(* CoDeSys 2.3 library: GermesLib_1_2.lib *)
(* Libraries: PID_Regulators.lib 6.11.19 15:29:27, Util.lib 18.5.10 15:14:28, STANDARD.LIB 4.10.05 11:14:46, IECSFC.LIB 13.4.06 15:51:28, ANALYZATION.LIB 5.10.99 09:05:06 *)

(* POU ChoosePumpRegime, CFC *)
FUNCTION_BLOCK ChoosePumpRegime
VAR
	pump1RStrig: RS;		(*Триггер-защелка выбора режима с главным первым насосом.*)
	pump2RStrig: RS;		(*Триггер-защелка выбора режима с главным вторым насосом.*)
	byCounterRStrig: RS;		(*Триггер-защелка выбора режима с запуском по количеству включений.*)
	byWorkTimeRStrig: RS;		(*Триггер-защелка выбора режима с запуском по наработке.*)
	Pump1MainDetector: R_TRIG;		(*Детектор переднего фронта включения режима, когда главный насос - первый.
Для сброса остальных значений.*)
	Pump2MainDetector: R_TRIG;		(*Детектор переднего фронта включения режима, когда главный насос - второй.
Для сброса остальных значений.*)
	ByCounterDetector: R_TRIG;		(*Детектор переднего фронта включения режима по количеству включений.
Для сброса остальных значений.*)
	ByWorkTimeDetector: R_TRIG;		(*Детектор переднего фронта включения режима по наработке.
Для сброса остальных значений.*)
END_VAR
VAR_INPUT
	start: BOOL;		(*Сигнал на включение насоса.
Активируется выход согласно выбранного режима.*)
	pump1Main: BOOL;		(*Режим: первый насос главный, второй - резервный.
Включать импульсом. Включать импульсом.*)
	pump2Main: BOOL;		(*Режим: второй насос главный, первый - резервный.
Включать импульсом. Включать импульсом.*)
	byCounter: BOOL;		(*Режим: запуск по количеству включений.
Включится с меньшим количеством стартов. Включать импульсом.*)
	byWorkTime: BOOL;		(*Режим: запуск по наработке.
Включится насос с меньшей наработкой. Включать импульсом.*)
END_VAR
VAR_OUTPUT
	pump1MainActive: BOOL;		(*Активный режим: первый насос главный.*)
	pump2MainActive: BOOL;		(*Активный режим: второй насос главный.*)
	byCounterActive: BOOL;		(*Активный режим: включение по количеству запусков.*)
	byWorkTimeActive: BOOL;		(*Активный режим: по наработке.*)
	startPump1: BOOL;		(*Запуск первого насоса как главного (основного).*)
	startPump2: BOOL;		(*Запуск второго насоса как главного (основного).*)
	startByCounter: BOOL;		(*Запуск насоса по количеству стартов.
			Запустится с меньшим. Если одинаково, то - первый.*)
	startByWorkTime: BOOL;		(*Запуск по наработке.
			Включится с меньшей. Если одинаково, то - первый.*)
END_VAR
VAR (* helpers for the ST form of the networks *)
	_en62 : BOOL;
	_t62 : BOOL;
	_en72 : BOOL;
	_t72 : BOOL;
	_en78 : BOOL;
	_t78 : BOOL;
	_en84 : BOOL;
	_t84 : BOOL;
END_VAR
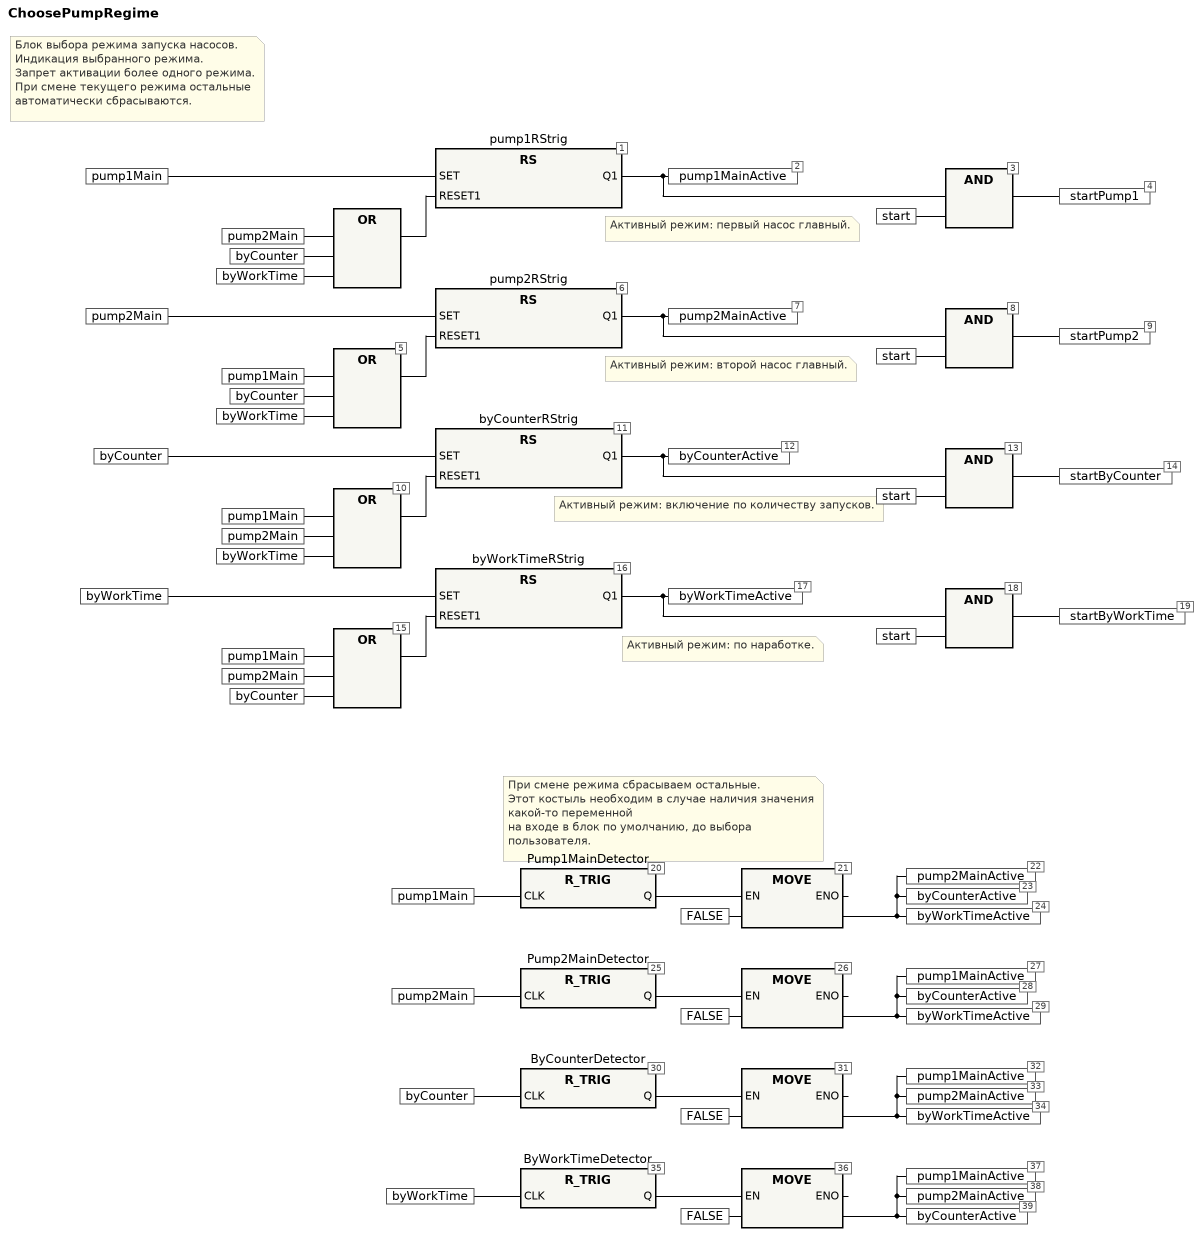
_CFC_ (* Continuous Function Chart, elements in execution order *)
(* При смене режима сбрасываем остальные. / Этот костыль необходим в случае наличия значения какой-то переменной / на входе в блок по умолчанию, до выбора пользователя. *)
(* Активный режим: второй насос главный. *)
(* Активный режим: по наработке. *)
(* Активный режим: включение по количеству запусков. *)
(* Активный режим: первый насос главный. *)
(* Блок выбора режима запуска насосов. / Индикация выбранного режима. / Запрет активации более одного режима. / При смене текущего режима остальные автоматически сбрасываются. *)
#0 OR(pump2Main, byCounter, byWorkTime)
#1 pump1RStrig:RS(SET: pump1Main, RESET1: #0)
#2 pump1MainActive <= #1.Q1
#3 AND(#1.Q1, start)
#4 startPump1 <= #3
#5 OR(pump1Main, byCounter, byWorkTime)
#6 pump2RStrig:RS(SET: pump2Main, RESET1: #5)
#7 pump2MainActive <= #6.Q1
#8 AND(#6.Q1, start)
#9 startPump2 <= #8
#10 OR(pump1Main, pump2Main, byWorkTime)
#11 byCounterRStrig:RS(SET: byCounter, RESET1: #10)
#12 byCounterActive <= #11.Q1
#13 AND(#11.Q1, start)
#14 startByCounter <= #13
#15 OR(pump1Main, pump2Main, byCounter)
#16 byWorkTimeRStrig:RS(SET: byWorkTime, RESET1: #15)
#17 byWorkTimeActive <= #16.Q1
#18 AND(#16.Q1, start)
#19 startByWorkTime <= #18
#20 Pump1MainDetector:R_TRIG(CLK: pump1Main)
#21 MOVE(EN: #20.Q, FALSE)
#22 pump2MainActive <= #21
#23 byCounterActive <= #21
#24 byWorkTimeActive <= #21
#25 Pump2MainDetector:R_TRIG(CLK: pump2Main)
#26 MOVE(EN: #25.Q, FALSE)
#27 pump1MainActive <= #26
#28 byCounterActive <= #26
#29 byWorkTimeActive <= #26
#30 ByCounterDetector:R_TRIG(CLK: byCounter)
#31 MOVE(EN: #30.Q, FALSE)
#32 pump1MainActive <= #31
#33 pump2MainActive <= #31
#34 byWorkTimeActive <= #31
#35 ByWorkTimeDetector:R_TRIG(CLK: byWorkTime)
#36 MOVE(EN: #35.Q, FALSE)
#37 pump1MainActive <= #36
#38 pump2MainActive <= #36
#39 byCounterActive <= #36
_END_CFC_
(* the same logic as Structured Text *)
(* При смене режима сбрасываем остальные. / Этот костыль необходим в случае наличия значения какой-то переменной / на входе в блок по умолчанию, до выбора пользователя. *)
(* Активный режим: второй насос главный. *)
(* Активный режим: по наработке. *)
(* Активный режим: включение по количеству запусков. *)
(* Активный режим: первый насос главный. *)
(* Блок выбора режима запуска насосов. / Индикация выбранного режима. / Запрет активации более одного режима. / При смене текущего режима остальные автоматически сбрасываются. *)
pump1RStrig(SET := pump1Main, RESET1 := pump2Main OR byCounter OR byWorkTime);
pump1MainActive := pump1RStrig.Q1;
startPump1 := pump1RStrig.Q1 AND start;
pump2RStrig(SET := pump2Main, RESET1 := pump1Main OR byCounter OR byWorkTime);
pump2MainActive := pump2RStrig.Q1;
startPump2 := pump2RStrig.Q1 AND start;
byCounterRStrig(SET := byCounter, RESET1 := pump1Main OR pump2Main OR byWorkTime);
byCounterActive := byCounterRStrig.Q1;
startByCounter := byCounterRStrig.Q1 AND start;
byWorkTimeRStrig(SET := byWorkTime, RESET1 := pump1Main OR pump2Main OR byCounter);
byWorkTimeActive := byWorkTimeRStrig.Q1;
startByWorkTime := byWorkTimeRStrig.Q1 AND start;
Pump1MainDetector(CLK := pump1Main);
_en62 := Pump1MainDetector.Q;
IF _en62 THEN _t62 := FALSE; END_IF;
IF _en62 THEN pump2MainActive := _t62; END_IF;
IF _en62 THEN byCounterActive := _t62; END_IF;
IF _en62 THEN byWorkTimeActive := _t62; END_IF;
Pump2MainDetector(CLK := pump2Main);
_en72 := Pump2MainDetector.Q;
IF _en72 THEN _t72 := FALSE; END_IF;
IF _en72 THEN pump1MainActive := _t72; END_IF;
IF _en72 THEN byCounterActive := _t72; END_IF;
IF _en72 THEN byWorkTimeActive := _t72; END_IF;
ByCounterDetector(CLK := byCounter);
_en78 := ByCounterDetector.Q;
IF _en78 THEN _t78 := FALSE; END_IF;
IF _en78 THEN pump1MainActive := _t78; END_IF;
IF _en78 THEN pump2MainActive := _t78; END_IF;
IF _en78 THEN byWorkTimeActive := _t78; END_IF;
ByWorkTimeDetector(CLK := byWorkTime);
_en84 := ByWorkTimeDetector.Q;
IF _en84 THEN _t84 := FALSE; END_IF;
IF _en84 THEN pump1MainActive := _t84; END_IF;
IF _en84 THEN pump2MainActive := _t84; END_IF;
IF _en84 THEN byCounterActive := _t84; END_IF;
END_FUNCTION_BLOCK

(* POU ControlAI, CFC *)
FUNCTION_BLOCK ControlAI
VAR_INPUT
	in: REAL;		(*Входное значение.*)
	minValue: REAL := 0;		(*Минимальное значение на выходе при 4мА на входе.
Если ко входу ничего не подключено, то 0.*)
	maxValue: REAL;		(*Максимальное значение на выходе при 20мА на входе.*)
END_VAR
VAR_OUTPUT
	out: REAL;		(*Выходное отфильтрованное значение.*)
	error: BOOL;		(*Ошибка входа.*)
END_VAR
VAR
	LIN_TRAFO: LIN_TRAFO;		(*Блок масштабирования входной величины.*)
	FilterREAL: FilterREAL;		(*Модуль фильтрации сигнала типа REAL.*)
END_VAR
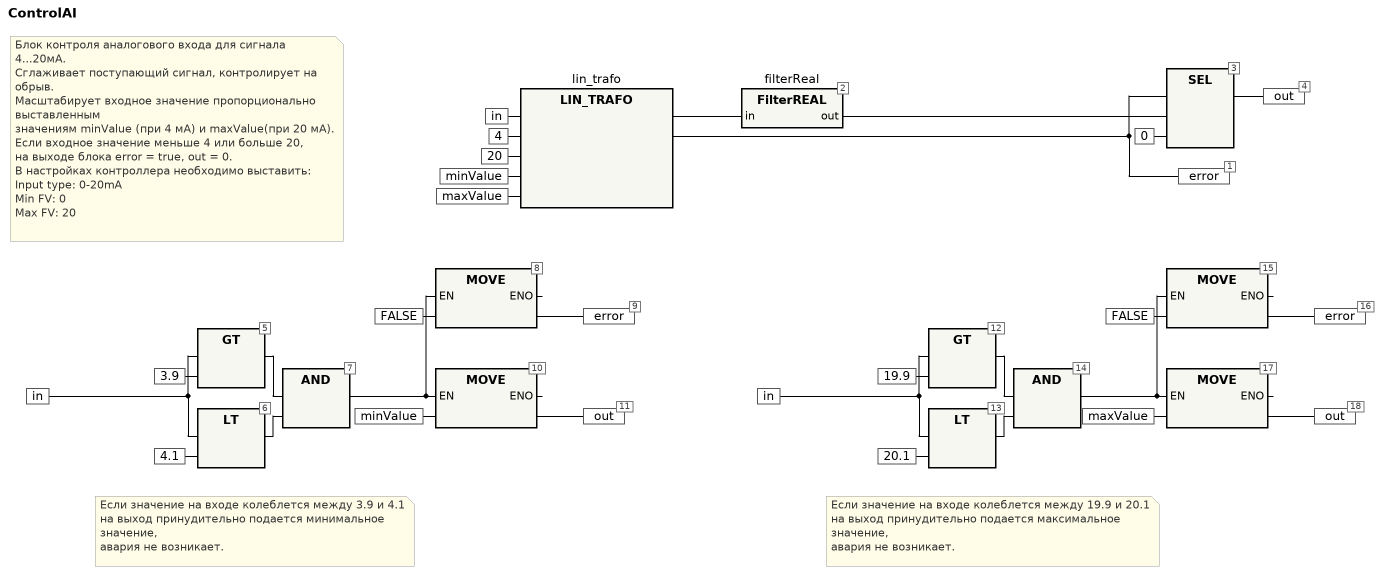
_CFC_ (* Continuous Function Chart, elements in execution order *)
(* Если значение на входе колеблется между 19.9 и 20.1 / на выход принудительно подается максимальное значение, / авария не возникает. *)
(* Если значение на входе колеблется между 3.9 и 4.1 / на выход принудительно подается минимальное значение, / авария не возникает. *)
(* Блок контроля аналогового входа для сигнала 4...20мА. / Сглаживает поступающий сигнал, контролирует на обрыв. / Масштабирует входное значение пропорционально выставленным / значениям minValue (при 4 мА) и maxValue(при 20 мА). / Если входное значение меньше 4 или больше 20, / на выходе блока error = true, out = 0. / В настройках контроллера необходимо выставить: / Input type: 0-20mA / Min FV: 0 / Max FV: 20 *)
#0 lin_trafo:LIN_TRAFO(in, 4, 20, minValue, maxValue)
#1 error <= #0.out 2
#2 filterReal:FilterREAL(in: #0.out 1)
#3 SEL(#0.out 2, #2.out, 0)
#4 out <= #3
#5 GT(in, 3.9)
#6 LT(in, 4.1)
#7 AND(#5, #6)
#8 MOVE(EN: #7, FALSE)
#9 error <= #8
#10 MOVE(EN: #7, minValue)
#11 out <= #10
#12 GT(in, 19.9)
#13 LT(in, 20.1)
#14 AND(#12, #13)
#15 MOVE(EN: #14, FALSE)
#16 error <= #15
#17 MOVE(EN: #14, maxValue)
#18 out <= #17
_END_CFC_
END_FUNCTION_BLOCK

(* POU FilterREAL, ST *)
FUNCTION_BLOCK FilterREAL
VAR_INPUT
	in: REAL; (*Входное значение*)
END_VAR
VAR_OUTPUT
	out: REAL; (*Выходное значение*)
END_VAR
VAR
	k: REAL; (*Коэффициент фильтра.Чем меньше тем плавнее, чем больше, тем быстрее работает фильтр.*)
END_VAR
(*Если разница между входом и выходом больше 0,5, то коэффициент большой, фильтр - быстрый, сглаживание - минимально.*)
IF ABS(in - out) > 0.01 THEN
	k := 0.9;
ELSE
	k:=0.0001;
END_IF
out := (in - out) * k + out;
END_FUNCTION_BLOCK

(* POU CounterManager, CFC *)
FUNCTION_BLOCK CounterManager

VAR
	pump1startsCounter: ImpulsCounter;		(*Счетчик количества включений насоса 1.*)
	pump2startsCounter: ImpulsCounter;		(*Счетчик количества включений насоса 2.*)
	counterRtrig: R_TRIG;		(*Детектор переднего фронта сигнала на запуск.*)
	counterFtrig: F_TRIG;		(*Детектор спада сигнала на запуск.*)
	counterRStrigPump1: RS;		(*RSтриггер сигнала на запуск насоса 1.*)
	counterRStrigPump2: RS;		(*RSтриггер сигнала на запуск насоса 2.*)
END_VAR
VAR_INPUT
	counterStart: BOOL;		(*Сигнал на запуск насоса с наименьшей наработкой.*)
	pump1ON: BOOL;		(*Сигнал подтверждение о запуске насоса 1.*)
	pump2ON: BOOL;		(*Сигнал подтверждение о запуске насоса 2.*)
	Pump1ResetCounter: BOOL;		(*Сброс счетчика включений насоса 1.*)
	Pump2ResetCounter: BOOL;		(*Сброс счетчика включений насоса 2.*)
END_VAR
VAR_OUTPUT
	counterPump1ON: BOOL;		(*Сигнал на запуск насоса 1.*)
	counterPump2ON: BOOL;		(*Сигнал на запуск насоса 2.*)
	counterPump1: DWORD;		(*Количество включений насоса 1.*)
	counterPump2: DWORD;		(*Количество включений насоса 2.*)
END_VAR
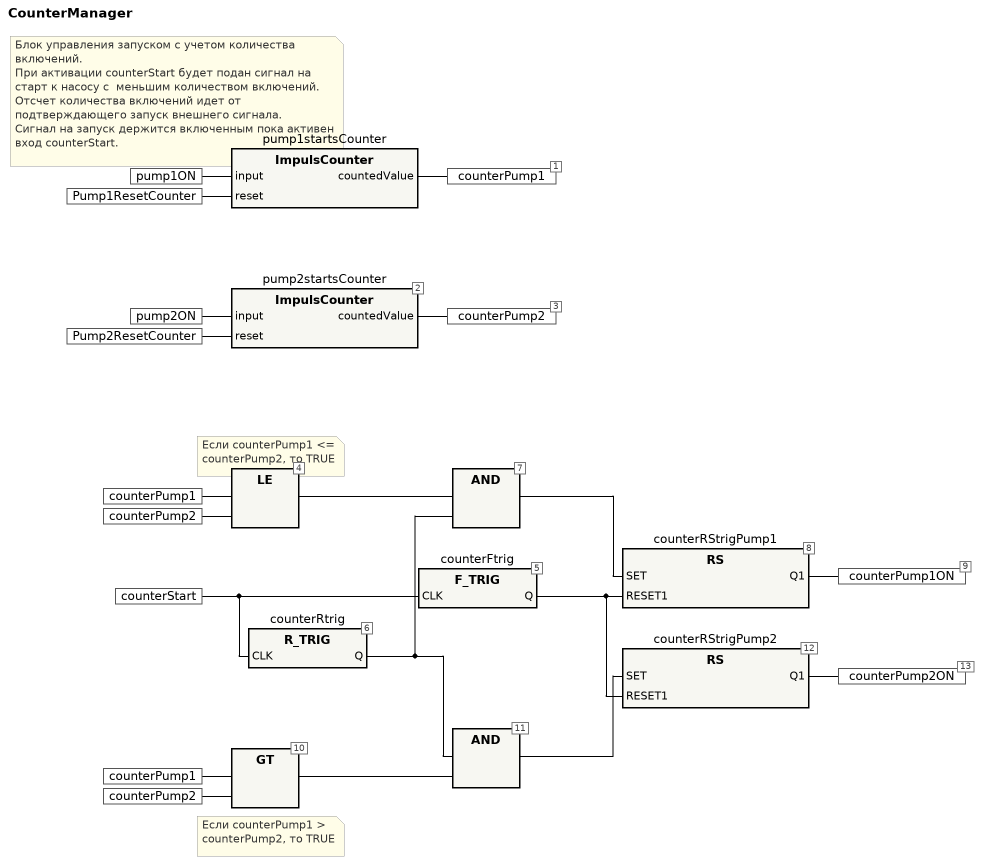
_CFC_ (* Continuous Function Chart, elements in execution order *)
(* Блок управления запуском с учетом количества включений. / При активации counterStart будет подан сигнал на старт к насосу с  меньшим количеством включений. / Отсчет количества включений идет от подтверждающего запуск внешнего сигнала. / Сигнал на запуск держится включенным пока активен вход counterStart. *)
(* Если counterPump1 <= / counterPump2, то TRUE *)
(* Если counterPump1 > / counterPump2, то TRUE *)
#0 pump1startsCounter:ImpulsCounter(input: pump1ON, reset: Pump1ResetCounter)
#1 counterPump1 <= #0.countedValue
#2 pump2startsCounter:ImpulsCounter(input: pump2ON, reset: Pump2ResetCounter)
#3 counterPump2 <= #2.countedValue
#4 LE(counterPump1, counterPump2)
#5 counterFtrig:F_TRIG(CLK: counterStart)
#6 counterRtrig:R_TRIG(CLK: counterStart)
#7 AND(#4, #6.Q)
#8 counterRStrigPump1:RS(SET: #7, RESET1: #5.Q)
#9 counterPump1ON <= #8.Q1
#10 GT(counterPump1, counterPump2)
#11 AND(#6.Q, #10)
#12 counterRStrigPump2:RS(SET: #11, RESET1: #5.Q)
#13 counterPump2ON <= #12.Q1
_END_CFC_
END_FUNCTION_BLOCK

(* POU ImpulsCounter, CFC *)
FUNCTION_BLOCK ImpulsCounter
VAR
	ImpulsDetector: R_TRIG;		(*Триггер переднего фронта входящего импульса.*)
END_VAR
VAR_INPUT
	input: BOOL;		(*Вход для импульсов, которые надо сосчитать.*)
	reset: BOOL;		(*Сброс счетчика.*)
END_VAR
VAR_OUTPUT
	countedValue: DWORD;		(*Суммарное количество импульсов.*)
END_VAR
VAR (* helpers for the ST form of the networks *)
	_t8 : DWORD;
END_VAR
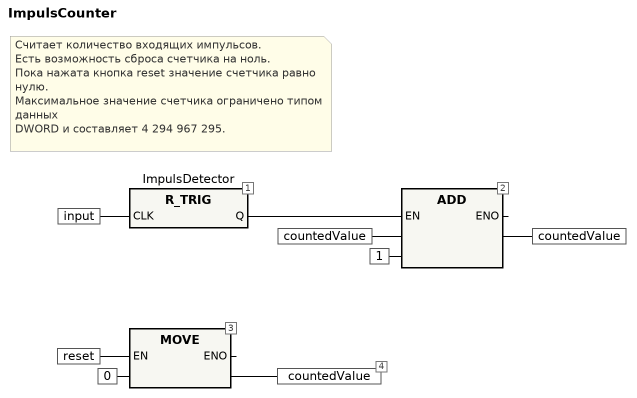
_CFC_ (* Continuous Function Chart, elements in execution order *)
(* Считает количество входящих импульсов. / Есть возможность сброса счетчика на ноль. / Пока нажата кнопка reset значение счетчика равно нулю. / Максимальное значение счетчика ограничено типом данных / DWORD и составляет 4 294 967 295. *)
#0 countedValue <= #2
#1 ImpulsDetector:R_TRIG(CLK: input)
#2 ADD(EN: #1.Q, countedValue, 1)
#3 MOVE(EN: reset, 0)
#4 countedValue <= #3
_END_CFC_
(* the same logic as Structured Text *)
(* Считает количество входящих импульсов. / Есть возможность сброса счетчика на ноль. / Пока нажата кнопка reset значение счетчика равно нулю. / Максимальное значение счетчика ограничено типом данных / DWORD и составляет 4 294 967 295. *)
countedValue := _t8;
ImpulsDetector(CLK := input);
IF ImpulsDetector.Q THEN _t8 := countedValue + 1; END_IF;
IF reset THEN countedValue := 0; END_IF;
END_FUNCTION_BLOCK

(* POU DosingPumpProportional, CFC *)
FUNCTION_BLOCK DosingPumpProportional
VAR_INPUT
	flowValue: REAL;		(*текущее значение мгновенного расхода, кубометров в час.*)
	setMinPumpDosingValue: REAL := 0;		(*задание минимальной производительности доз.насоса.
По умолчанию, если ничего не подключено ко входу, равно нулю.*)
	setMaxPumpDosingValue: REAL;		(*задание максимальной производительности доз.насоса, в мл/мин*)
	minOutputValue: REAL := 4;		(*минимальное значение выходного сигнала.
По умолчанию, если ничего не подключено ко входу, равно 4.*)
	maxOutputValue: REAL := 20;		(*Максимально значение выходного сигнала.
По умолчанию, если ничего не подключено ко входу, равно 20.*)
	setKoeffProportionality: REAL;		(*Задание мл на кубометр (коэф.пропорциональности между расходом и дозированием)*)
	minFlowToStart: REAL := 10;		(*Минимальное значение расхода для подачи сигнала на начало дозирования.
По умолчанию, если ничего не подключено ко входу, равно 10 кубометров в час.*)
END_VAR
VAR_OUTPUT
	outputValue: REAL;		(*Выходной сигнал на дозирующий насос.*)
	dosingError: BOOL;		(*Ошибка производительности дозирования (неверно заданы значения производительности насоса, производительность доз.насоса не соответствует расходу.*)
	startDosingPump: BOOL;		(*Сигнал на запуск дозирующего насоса.*)
END_VAR
VAR
	linearTransformator: LIN_TRAFO;		(*получает на вход значение из указанного диапазона, ставит на выходе пропорциональное значение из другого диапазона.*)
END_VAR
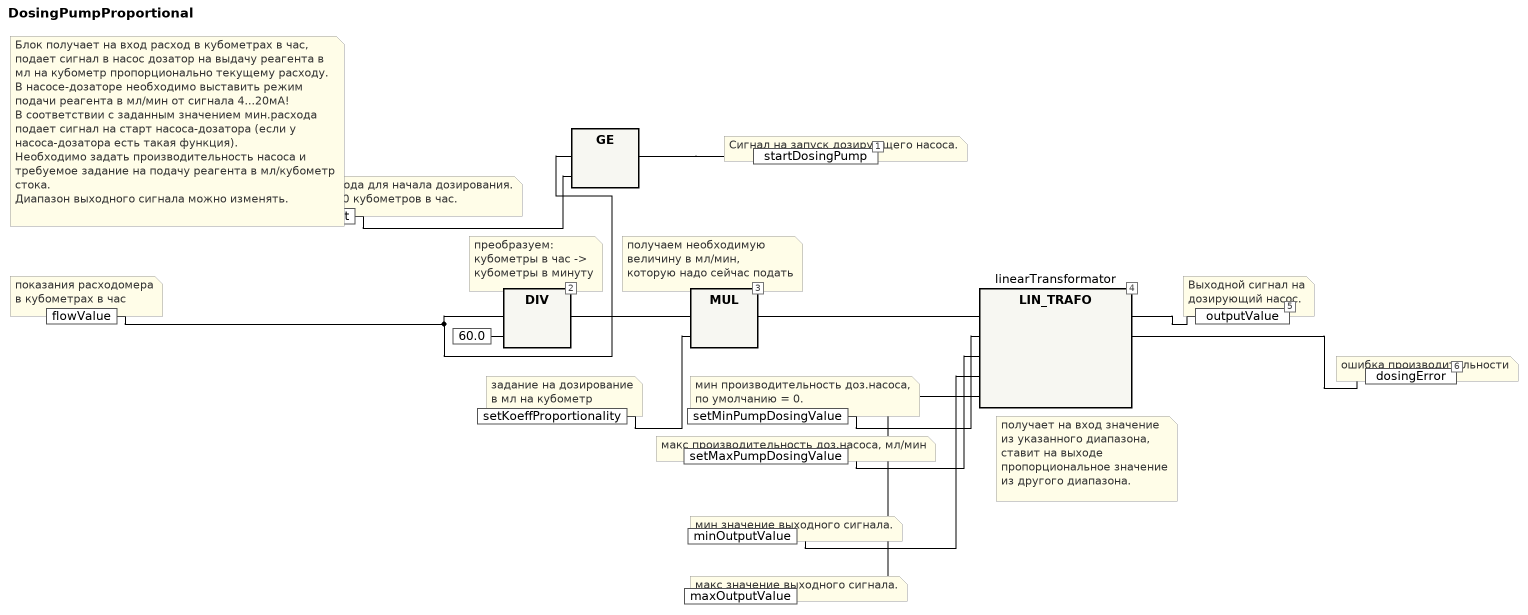
_CFC_ (* Continuous Function Chart, elements in execution order *)
(* Сигнал на запуск дозирующего насоса. *)
(* min значение расхода для начала дозирования. / По умолчанию = 10 кубометров в час. *)
(* макс производительность доз.насоса, мл/мин *)
(* мин производительность доз.насоса, / по умолчанию = 0. *)
(* получаем необходимую / величину в мл/мин, / которую надо сейчас подать *)
(* задание на дозирование / в мл на кубометр *)
(* показания расходомера / в кубометрах в час *)
(* преобразуем: / кубометры в час -> / кубометры в минуту *)
(* мин значение выходного сигнала. *)
(* макс значение выходного сигнала. *)
(* Выходной сигнал на / дозирующий насос. *)
(* ошибка производительности *)
(* получает на вход значение / из указанного диапазона, / ставит на выходе / пропорциональное значение / из другого диапазона. *)
(* Блок получает на вход расход в кубометрах в час, подает сигнал в насос дозатор на выдачу реагента в мл на кубометр пропорционально текущему расходу. / В насосе-дозаторе необходимо выставить режим подачи реагента в мл/мин от сигнала 4...20мА! / В соответствии с заданным значением мин.расхода подает сигнал на старт насоса-дозатора (если у насоса-дозатора есть такая функция). / Необходимо задать производительность насоса и требуемое задание на подачу реагента в мл/кубометр стока. / Диапазон выходного сигнала можно изменять. *)
#0 GE(flowValue, minFlowToStart)
#1 startDosingPump <= #0
#2 DIV(flowValue, 60.0)
#3 MUL(#2, setKoeffProportionality)
#4 linearTransformator:LIN_TRAFO(#3, setMinPumpDosingValue, setMaxPumpDosingValue, minOutputValue, maxOutputValue)
#5 outputValue <= #4.out 1
#6 dosingError <= #4.out 2
_END_CFC_
END_FUNCTION_BLOCK

(* POU FlowVolume, CFC *)
FUNCTION_BLOCK FlowVolume
VAR_INPUT
	flowValue: REAL;		(*Вход от расходомера, мгновенный расход в кубометрах в час.*)
	setVolume: REAL;		(*Контрольный объем. Сравнивается с накопленным по показаниям расходомера,
Если превышает, счетчик сбрасывается, на выход out подается импульс.
Если на входе ноль, то условие не работает, блок просто считает сумму стоков.*)
	reset: BOOL;		(*Ручной сброс счетчика.*)
END_VAR
VAR_OUTPUT
	totalAmount: REAL;		(*Сумма накопленных стоков.*)
	out: BOOL;		(*Импульс - сигнал что сумма стоков равна или больше
заданному в setVolume значению.*)
END_VAR
VAR
	pulsPerSec: PulsePerSec;		(*Генератор импульс в секунду.*)
END_VAR
VAR (* helpers for the ST form of the networks *)
	_t22 : BOOL;
END_VAR
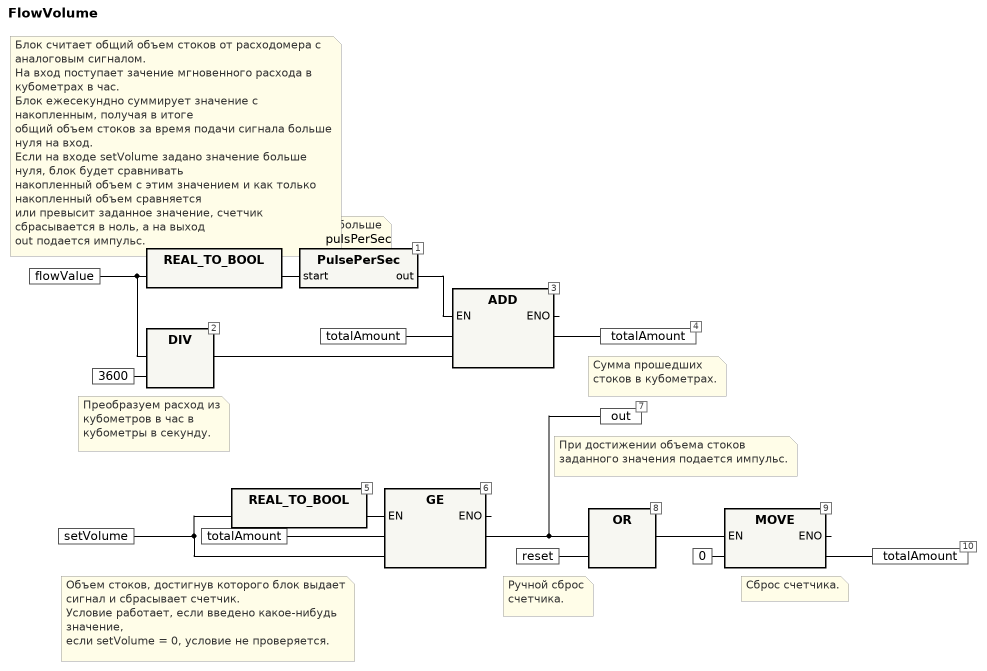
_CFC_ (* Continuous Function Chart, elements in execution order *)
(* Ручной сброс / счетчика. *)
(* При достижении объема стоков / заданного значения подается импульс. *)
(* Сумма прошедших / стоков в кубометрах. *)
(* Объем стоков, достигнув которого блок выдает / сигнал и сбрасывает счетчик. / Условие работает, если введено какое-нибудь значение, / если setVolume = 0, условие не проверяется. *)
(* Преобразуем расход из / кубометров в час в / кубометры в секунду. *)
(* Начинаем считать стоки при наличии расхода больше нуля. *)
(* Сброс счетчика. *)
(* Блок считает общий объем стоков от расходомера с аналоговым сигналом. / На вход поступает зачение мгновенного расхода в кубометрах в час. / Блок ежесекундно суммирует значение с накопленным, получая в итоге / общий объем стоков за время подачи сигнала больше нуля на вход. / Если на входе setVolume задано значение больше нуля, блок будет сравнивать / накопленный объем с этим значением и как только накопленный объем сравняется / или превысит заданное значение, счетчик сбрасывается в ноль, а на выход / out подается импульс. *)
#0 REAL_TO_BOOL(flowValue)
#1 pulsPerSec:PulsePerSec(start: #0)
#2 DIV(flowValue, 3600)
#3 ADD(EN: #1.out, totalAmount, #2)
#4 totalAmount <= #3
#5 REAL_TO_BOOL(setVolume)
#6 GE(EN: #5, totalAmount, setVolume)
#7 out <= #6
#8 OR(#6, reset)
#9 MOVE(EN: #8, 0)
#10 totalAmount <= #9
_END_CFC_
(* the same logic as Structured Text *)
(* Ручной сброс / счетчика. *)
(* При достижении объема стоков / заданного значения подается импульс. *)
(* Сумма прошедших / стоков в кубометрах. *)
(* Объем стоков, достигнув которого блок выдает / сигнал и сбрасывает счетчик. / Условие работает, если введено какое-нибудь значение, / если setVolume = 0, условие не проверяется. *)
(* Преобразуем расход из / кубометров в час в / кубометры в секунду. *)
(* Начинаем считать стоки при наличии расхода больше нуля. *)
(* Сброс счетчика. *)
(* Блок считает общий объем стоков от расходомера с аналоговым сигналом. / На вход поступает зачение мгновенного расхода в кубометрах в час. / Блок ежесекундно суммирует значение с накопленным, получая в итоге / общий объем стоков за время подачи сигнала больше нуля на вход. / Если на входе setVolume задано значение больше нуля, блок будет сравнивать / накопленный объем с этим значением и как только накопленный объем сравняется / или превысит заданное значение, счетчик сбрасывается в ноль, а на выход / out подается импульс. *)
pulsPerSec(start := REAL_TO_BOOL(flowValue));
IF pulsPerSec.out THEN totalAmount := totalAmount + (flowValue / 3600); END_IF;
IF REAL_TO_BOOL(setVolume) THEN _t22 := totalAmount >= setVolume; END_IF;
out := _t22;
IF _t22 OR reset THEN totalAmount := 0; END_IF;
END_FUNCTION_BLOCK

(* POU PulsePerSec, CFC *)
FUNCTION_BLOCK PulsePerSec
VAR_INPUT
	start: BOOL;		(*Включает генератор импульсов.*)
END_VAR
VAR_OUTPUT
	out: BOOL;		(*Выход генератора импульсов. Начинает с FALSE.
			Каждую секунду выдает BOOL: TRUE.*)
END_VAR
VAR
	pulserRtrig: R_TRIG;		(*Детектор переднего фронта подачи импульсов.*)
	pulserRTC: RTC;		(*Таймер реального времени.*)
END_VAR
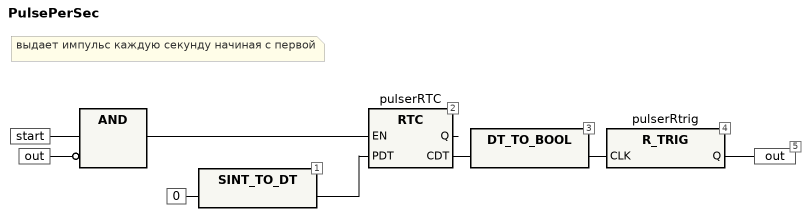
_CFC_ (* Continuous Function Chart, elements in execution order *)
(* выдает импульс каждую секунду начиная с первой *)
#0 AND(start, NOT out)
#1 SINT_TO_DT(0)
#2 pulserRTC:RTC(EN: #0, PDT: #1)
#3 DT_TO_BOOL(#2.CDT)
#4 pulserRtrig:R_TRIG(CLK: #3)
#5 out <= #4.Q
_END_CFC_
(* the same logic as Structured Text *)
(* выдает импульс каждую секунду начиная с первой *)
pulserRTC(EN := start AND NOT out, PDT := SINT_TO_DT(0));
pulserRtrig(CLK := DT_TO_BOOL(pulserRTC.CDT));
out := pulserRtrig.Q;
END_FUNCTION_BLOCK

(* POU IfBOOL, ST *)
FUNCTION_BLOCK IfBOOL
VAR_INPUT
	key: BOOL; (*Ключ. Если TRUE, то сигнал на входе будет передан на выход keyTRUE, иначе на keyFALSE.*)
	input: BOOL; (*Вход*)
END_VAR
VAR_OUTPUT
	keyFALSE: BOOL; (*Выход  получит значение от входа, если key = FALSE.*)
	keyTRUE: BOOL; (*Выход  получит значение от входа, если key = TRUE.*)
END_VAR
VAR
END_VAR
IF key = TRUE THEN
	keyTRUE := input;
	keyFALSE := FALSE;
ELSE keyTRUE := FALSE;
		keyFALSE := input;
END_IF
END_FUNCTION_BLOCK

(* POU ImpulsFlowCounter, CFC *)
FUNCTION_BLOCK ImpulsFlowCounter
VAR_INPUT
	impulsInput: BOOL;		(*Входящие импульсы от расходомера.
Каждый импульс будет прибавлять в итоговую сумму величину веса импульса.*)
	impulsValue: REAL;		(*Вес импульса расходомера.*)
	resetCounter: BOOL;		(*Сброс счетчика.*)
	correctionValue: REAL;		(*Число, которое будет прибавлено или вычтено из накопленной суммы.*)
	addCorrection: BOOL;		(*Прибавить коррекцию к накопленной сумме.*)
	deleteCorrection: BOOL;		(*Вычесть коррекцию из накопленной суммы.
Если получится отрицательное число, сумма скинется в ноль.*)
END_VAR
VAR_OUTPUT
	totalAmountREAL: REAL;		(*Накопленная сумма в десятичном виде.
От 10 млн может выводиться в экспоненциальной форме.*)
	totalAmountDWORD: DWORD;		(*Накопленная сумма в целочисленном виде.
Округление десятичных по правилам арифметики.*)
END_VAR
VAR
	inputImpulsRtrig: R_TRIG;		(*Детектор переднего фронта входящих импульсов.*)
	resetRtrig: R_TRIG;		(*Детектор переднего фронта сигнала на сброс счетчика.*)
	addCorrRtrig: R_TRIG;		(*Детектор переднего фронта сигнала на прибавление коррекции.*)
	deleteCorrRtrig: R_TRIG;		(*Детектор переднего фронта сигнала на вычитание коррекции.*)
END_VAR
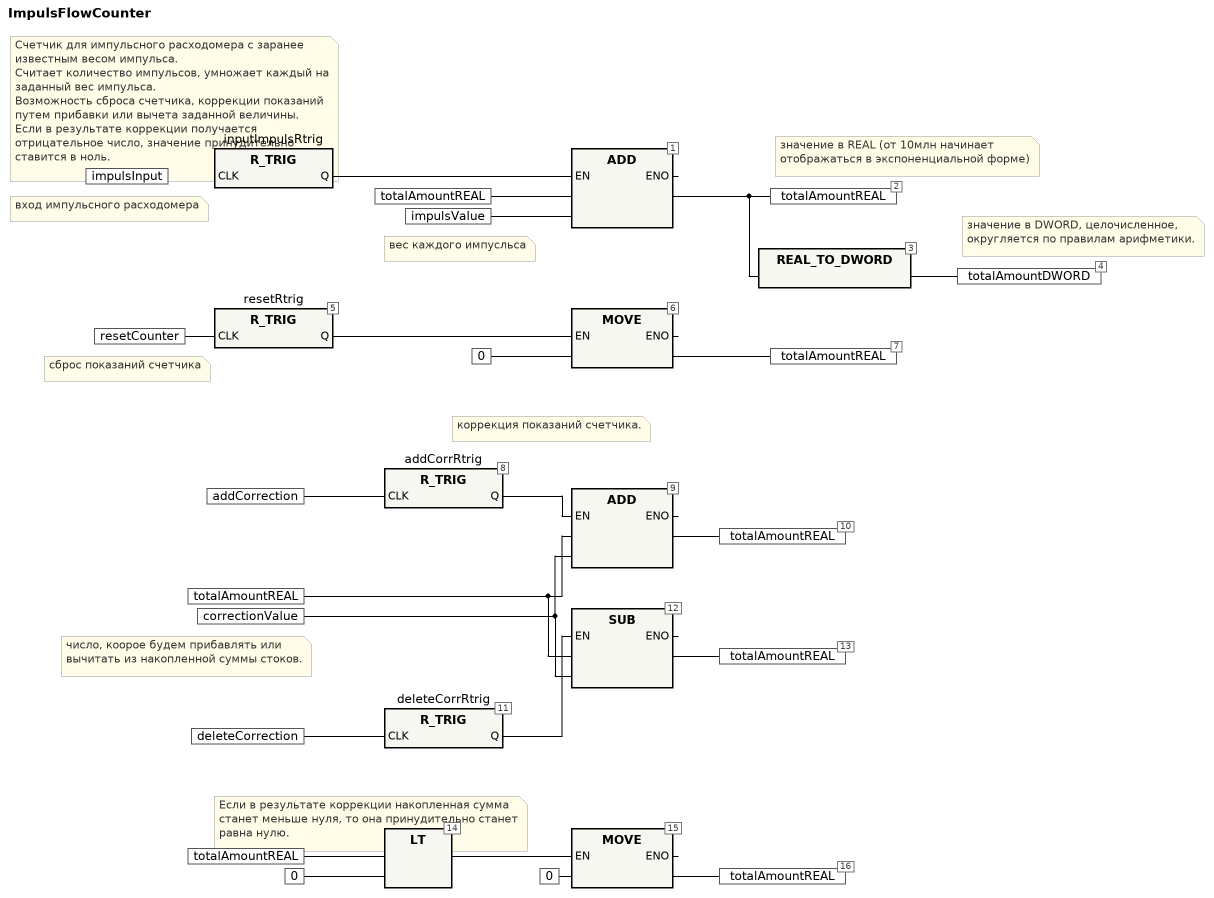
_CFC_ (* Continuous Function Chart, elements in execution order *)
(* вход импульсного расходомера *)
(* сброс показаний счетчика *)
(* значение в REAL (от 10млн начинает / отображаться в экспоненциальной форме) *)
(* значение в DWORD, целочисленное, / округляется по правилам арифметики. *)
(* Если в результате коррекции накопленная сумма станет меньше нуля, то она принудительно станет равна нулю. *)
(* коррекция показаний счетчика. *)
(* число, коорое будем прибавлять или / вычитать из накопленной суммы стоков. *)
(* вес каждого импусльса *)
(* Счетчик для импульсного расходомера с заранее известным весом импульса. / Считает количество импульсов, умножает каждый на заданный вес импульса. / Возможность сброса счетчика, коррекции показаний путем прибавки или вычета заданной величины. / Если в результате коррекции получается отрицательное число, значение принудительно ставится в ноль. *)
#0 inputImpulsRtrig:R_TRIG(CLK: impulsInput)
#1 ADD(EN: #0.Q, totalAmountREAL, impulsValue)
#2 totalAmountREAL <= #1
#3 REAL_TO_DWORD(#1)
#4 totalAmountDWORD <= #3
#5 resetRtrig:R_TRIG(CLK: resetCounter)
#6 MOVE(EN: #5.Q, 0)
#7 totalAmountREAL <= #6
#8 addCorrRtrig:R_TRIG(CLK: addCorrection)
#9 ADD(EN: #8.Q, totalAmountREAL, correctionValue)
#10 totalAmountREAL <= #9
#11 deleteCorrRtrig:R_TRIG(CLK: deleteCorrection)
#12 SUB(EN: #11.Q, totalAmountREAL, correctionValue)
#13 totalAmountREAL <= #12
#14 LT(totalAmountREAL, 0)
#15 MOVE(EN: #14, 0)
#16 totalAmountREAL <= #15
_END_CFC_
END_FUNCTION_BLOCK

(* POU QueueManager, CFC *)
FUNCTION_BLOCK QueueManager
VAR_INPUT
	input: BOOL;		(*Вход сигнала на регенерацию.*)
	testValves: BOOL;		(*Тест заслонок. Имитирует подачу сигнала на регенерацию.*)
	filterAlarm: BOOL;		(*Сигнал авария от управляющего клапана.*)
	regenFilterStatus: BOOL;		(*Сигнал от управляющего клапана о текущем режиме.*)
	alarmReset: BOOL;		(*Сброс аварий.*)
	startNextLoop: BOOL;		(*Запуск нового цикла регенерации. Все сигналы о том, что фильтры
отрегенерированы сбрасываются.*)
	filterValveOpened: BOOL;		(*Заслонка фильтрации открыта.*)
	filterValveClosed: BOOL;		(*Заслонка фильтрации закрыта.*)
	regenValveOpened: BOOL;		(*Заслонка регенерации открыта.*)
	regenValveClosed: BOOL;		(*Заслонка регенерации закрыта.*)
	timeToOpenClose: WORD;		(*Время на открытие/закрытие заслонки в секундах.*)
END_VAR
VAR_OUTPUT
	output: BOOL;		(*Выход для связи с остальными блоками управления очередью
на промывку. В последнем не подключается.*)
	filterValveToOpen: BOOL;		(*Открыть заслонку фильтрации.*)
	filterValveToClose: BOOL;		(*Закрыть заслонку фильтрации.*)
	errorToOpenFilterValve: BOOL;		(*Заслонка фильтрации не открылась за заданное время.*)
	errorToCloseFilterValve: BOOL;		(*Заслонка фильтрации не закрылась за заданное время.*)
	regenValveToOpen: BOOL;		(*Открыть заслонку регенерации.*)
	regenValveToClose: BOOL;		(*Закрыть заслонку регенерации.*)
	errorToOpenRegenValve: BOOL;		(*Заслонка регенерации не открылась за заданное время.*)
	errorToCloseRegenValve: BOOL;		(*Заслонка регенерации не закрылась за заданное время.*)
	regenerated: BOOL;		(*Фильтр прошел регенерацию.*)
	failToRegen: BOOL;		(*Попытка регенерации не удалась.*)
	loopFinished: BOOL;		(*Вход последнего блока подключить во входы startNextLoop во всех блоках,
включая самого себя. В остальных блоках выход не задействовать.*)
	startRegen: BOOL; (*Команда на промывку фильтра*)
END_VAR
VAR
	valveAlarm: BOOL;		(*Общий сигнал авария от обеих заслонок.*)
	QueueModule: QueueModule;		(*Модуль управления очередью на регенерацию.*)
	filterValve: SimpleValve;		(*Блок управления заслонкой фильтрации.*)
	regenrValve: SimpleValve;		(*Блок управления заслонкой регенерации.*)
END_VAR
VAR (* helpers for the ST form of the networks *)
	_t21 : BOOL;
END_VAR
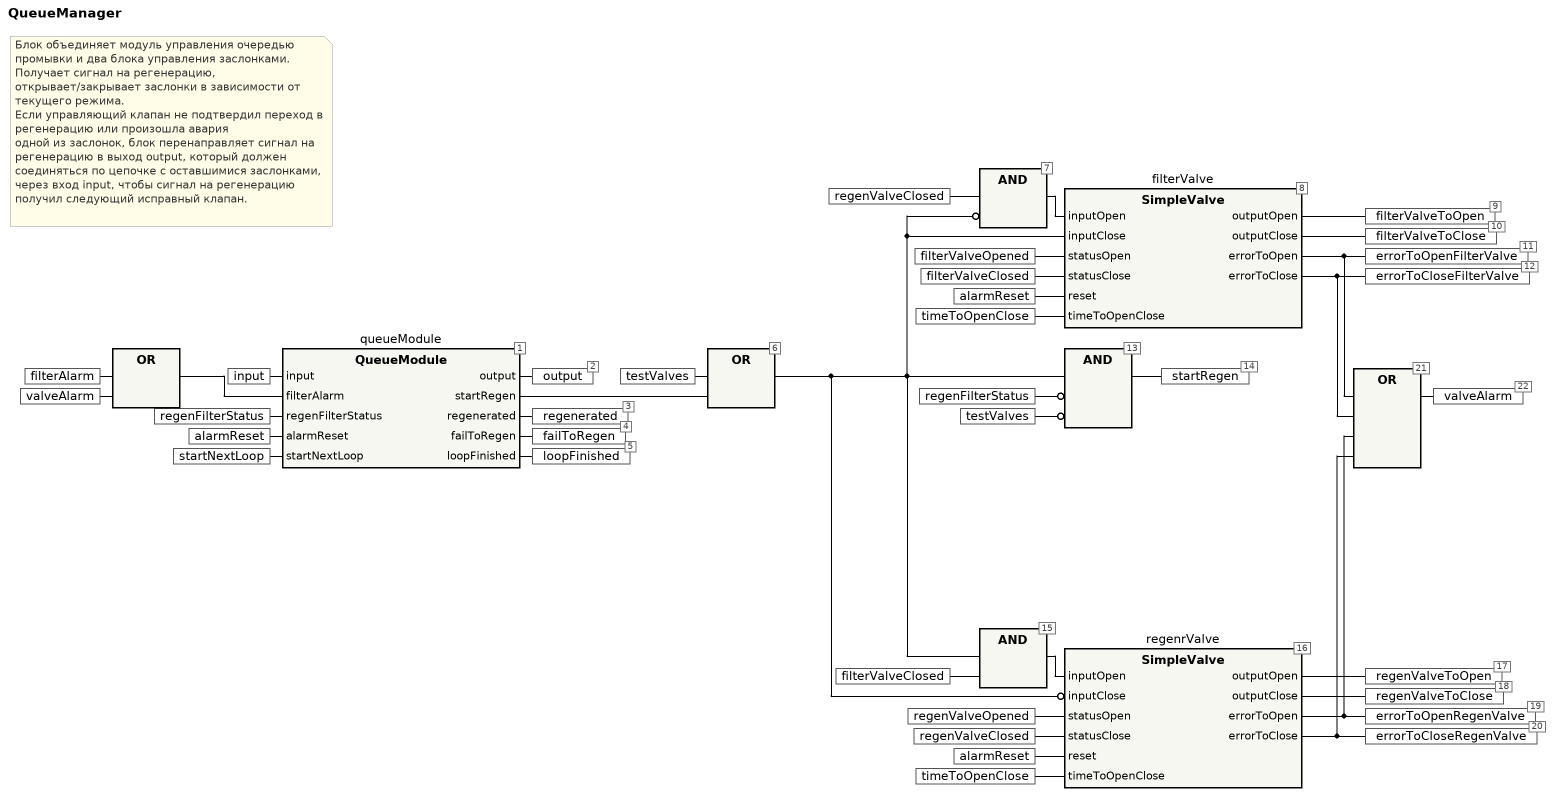
_CFC_ (* Continuous Function Chart, elements in execution order *)
(* Блок объединяет модуль управления очередью промывки и два блока управления заслонками. / Получает сигнал на регенерацию, открывает/закрывает заслонки в зависимости от текущего режима. / Если управляющий клапан не подтвердил переход в регенерацию или произошла авария / одной из заслонок, блок перенаправляет сигнал на регенерацию в выход output, который должен / соединяться по цепочке с оставшимися заслонками, через вход input, чтобы сигнал на регенерацию / получил следующий исправный клапан. *)
#0 OR(filterAlarm, valveAlarm)
#1 queueModule:QueueModule(input: input, filterAlarm: #0, regenFilterStatus: regenFilterStatus, alarmReset: alarmReset, startNextLoop: startNextLoop)
#2 output <= #1.output
#3 regenerated <= #1.regenerated
#4 failToRegen <= #1.failToRegen
#5 loopFinished <= #1.loopFinished
#6 OR(testValves, #1.startRegen)
#7 AND(regenValveClosed, NOT #6)
#8 filterValve:SimpleValve(inputOpen: #7, inputClose: #6, statusOpen: filterValveOpened, statusClose: filterValveClosed, reset: alarmReset, timeToOpenClose: timeToOpenClose)
#9 filterValveToOpen <= #8.outputOpen
#10 filterValveToClose <= #8.outputClose
#11 errorToOpenFilterValve <= #8.errorToOpen
#12 errorToCloseFilterValve <= #8.errorToClose
#13 AND(#6, NOT regenFilterStatus, NOT testValves)
#14 startRegen <= #13
#15 AND(#6, filterValveClosed)
#16 regenrValve:SimpleValve(inputOpen: #15, inputClose: NOT #6, statusOpen: regenValveOpened, statusClose: regenValveClosed, reset: alarmReset, timeToOpenClose: timeToOpenClose)
#17 regenValveToOpen <= #16.outputOpen
#18 regenValveToClose <= #16.outputClose
#19 errorToOpenRegenValve <= #16.errorToOpen
#20 errorToCloseRegenValve <= #16.errorToClose
#21 OR(#8.errorToOpen, #8.errorToClose, #16.errorToOpen, #16.errorToClose)
#22 valveAlarm <= #21
_END_CFC_
(* the same logic as Structured Text *)
(* Блок объединяет модуль управления очередью промывки и два блока управления заслонками. / Получает сигнал на регенерацию, открывает/закрывает заслонки в зависимости от текущего режима. / Если управляющий клапан не подтвердил переход в регенерацию или произошла авария / одной из заслонок, блок перенаправляет сигнал на регенерацию в выход output, который должен / соединяться по цепочке с оставшимися заслонками, через вход input, чтобы сигнал на регенерацию / получил следующий исправный клапан. *)
queueModule(input := input, filterAlarm := filterAlarm OR valveAlarm, regenFilterStatus := regenFilterStatus, alarmReset := alarmReset, startNextLoop := startNextLoop);
output := queueModule.output;
regenerated := queueModule.regenerated;
failToRegen := queueModule.failToRegen;
loopFinished := queueModule.loopFinished;
_t21 := testValves OR queueModule.startRegen;
filterValve(inputOpen := regenValveClosed AND NOT _t21, inputClose := _t21, statusOpen := filterValveOpened, statusClose := filterValveClosed, reset := alarmReset, timeToOpenClose := timeToOpenClose);
filterValveToOpen := filterValve.outputOpen;
filterValveToClose := filterValve.outputClose;
errorToOpenFilterValve := filterValve.errorToOpen;
errorToCloseFilterValve := filterValve.errorToClose;
startRegen := _t21 AND NOT regenFilterStatus AND NOT testValves;
regenrValve(inputOpen := _t21 AND filterValveClosed, inputClose := NOT _t21, statusOpen := regenValveOpened, statusClose := regenValveClosed, reset := alarmReset, timeToOpenClose := timeToOpenClose);
regenValveToOpen := regenrValve.outputOpen;
regenValveToClose := regenrValve.outputClose;
errorToOpenRegenValve := regenrValve.errorToOpen;
errorToCloseRegenValve := regenrValve.errorToClose;
valveAlarm := filterValve.errorToOpen OR filterValve.errorToClose OR regenrValve.errorToOpen OR regenrValve.errorToClose;
END_FUNCTION_BLOCK

(* POU QueueModule, CFC *)
FUNCTION_BLOCK QueueModule
VAR_INPUT
	input: BOOL;		(*Вход на старт регенерации.*)
	filterAlarm: BOOL;		(*Вход аварии от управляющего клапана фильтра.*)
	regenFilterStatus: BOOL;		(*Вход для сигнала подтверждения начала регенерации
от фильтра.*)
	alarmReset: BOOL;		(*Сброс статуса о неудачной попытке регенерации.*)
	startNextLoop: BOOL;		(*Запустить новый цикл, сбрасываются все статусы промытости
фильтров, начало снова от первого фильтра.*)
END_VAR
VAR_OUTPUT
	output: BOOL;		(*Выход, передающий сигнал от счетчика о начале регенерации,
на следующий фильтр. Соединять с input следующего блока, если он есть.*)
	startRegen: BOOL;		(*Выход на старт регенерации, подаваемый на фильтр.*)
	regenerated: BOOL;		(*TRUE, если этот фильтр уже промыт.*)
	failToRegen: BOOL;		(*Не удалось запустить регенерацию.
Не пришло подтверждение от фильтра более 5 сек после старта.*)
	loopFinished: BOOL;		(*Импульсный сигнал, возникающий при отключени сигнала подтверждения
статуса промывки от фильтра (фильтр вернулся в режим фильтрации) или при неудачной попытке регенерации. 
Использовать в последнем блоке для старта нового цикла во всех блоках.*)
END_VAR
VAR
	regStatusDelay: TON;		(*Таймер задержки ожидания подтверждения от фильтра
о начале регенерации.*)
	regStartRS: RS;		(*Триггер старта регенерации.*)
	failureRS: RS;		(*Триггер неудачного пуска регенерации.*)
	successRS: RS;		(*Триггер удачной регенерации.*)
	regenFilterOFF: F_TRIG;		(*Триггер контроля отключения сигнала от фильтра, что он закончил
режим промывки для возврата задвижек обратно в режим фильтрации.*)
	failureRtrig: R_TRIG;		(*детектор переднего фронта сигнала о неудачной попытке регенерации.*)
END_VAR
VAR (* helpers for the ST form of the networks *)
	_t45 : BOOL;
	_t78 : BOOL;
END_VAR
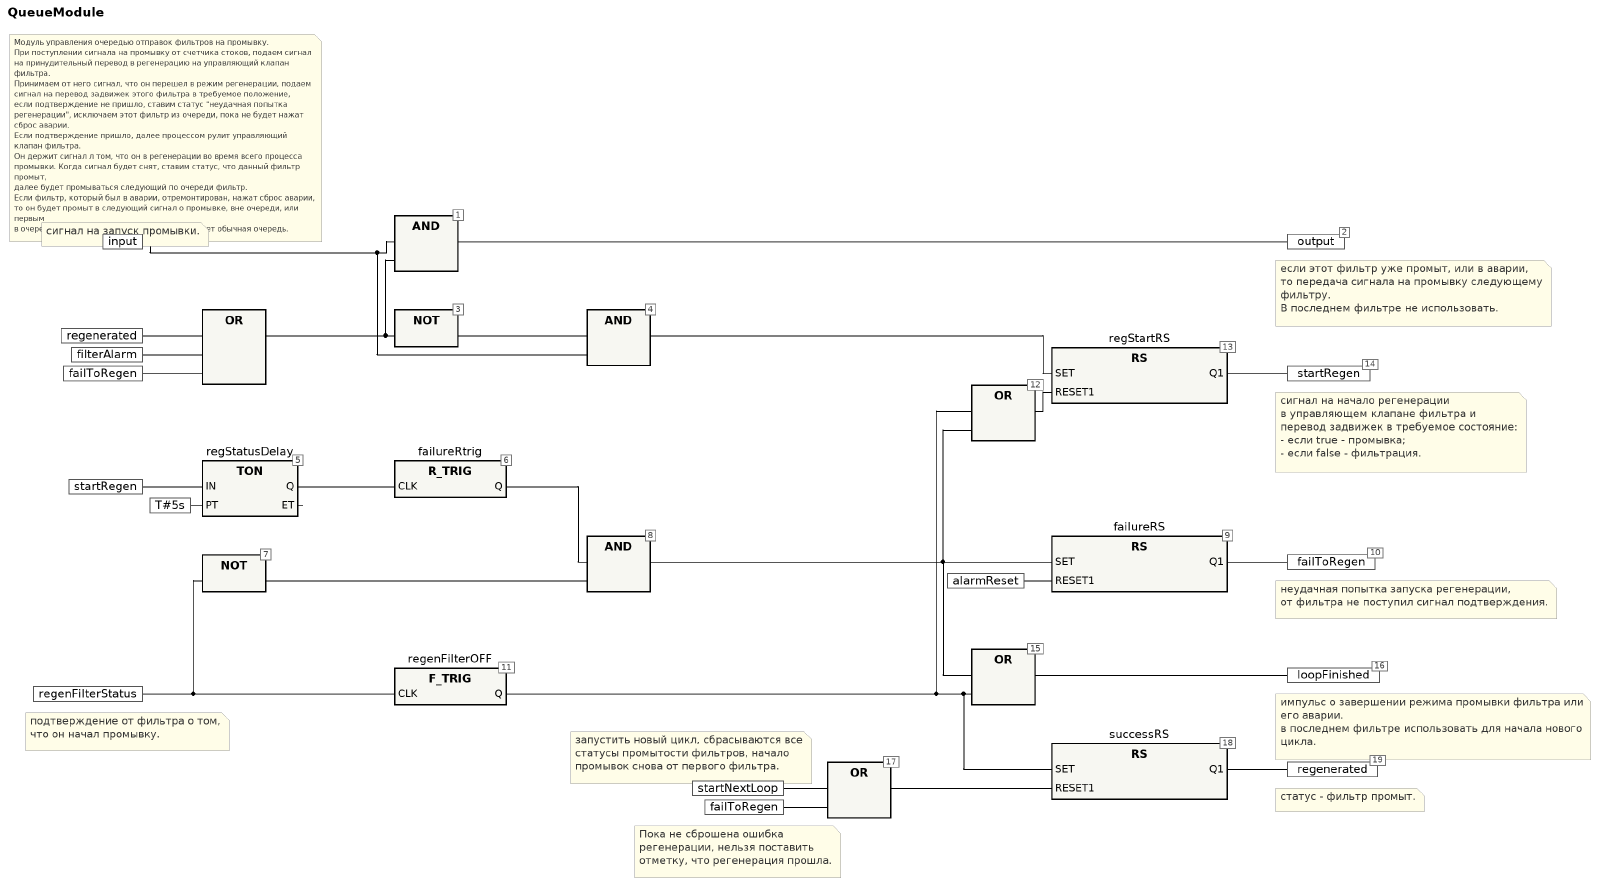
_CFC_ (* Continuous Function Chart, elements in execution order *)
(* Пока не сброшена ошибка / регенерации, нельзя поставить / отметку, что регенерация прошла. *)
(* запустить новый цикл, сбрасываются все / статусы промытости фильтров, начало / промывок снова от первого фильтра. *)
(* Модуль управления очередью отправок фильтров на промывку. / При поступлении сигнала на промывку от счетчика стоков, подаем сигнал на принудительный перевод в регенерацию на управляющий клапан фильтра. / Принимаем от него сигнал, что он перешел в режим регенерации, подаем сигнал на перевод задвижек этого фильтра в требуемое положение, / если подтверждение не пришло, ставим статус "неудачная попытка регенерации", исключаем этот фильтр из очереди, пока не будет нажат сброс аварии. / Если подтверждение пришло, далее процессом рулит управляющий клапан фильтра. / Он держит сигнал л том, что он в регенерации во время всего процесса промывки. Когда сигнал будет снят, ставим статус, что данный фильтр промыт, / далее будет промываться следующий по очереди фильтр. / Если фильтр, который был в аварии, отремонтирован, нажат сброс аварии, то он будет промыт в следующий сигнал о промывке, вне очереди, или первым / в очереди отремонтированных, после чего пойдет обычная очередь. *)
(* сигнал на запуск промывки. *)
(* если этот фильтр уже промыт, или в аварии, / то передача сигнала на промывку следующему фильтру. / В последнем фильтре не использовать. *)
(* сигнал на начало регенерации / в управляющем клапане фильтра и / перевод задвижек в требуемое состояние: / - если true - промывка; / - если false - фильтрация. *)
(* неудачная попытка запуска регенерации, / от фильтра не поступил сигнал подтверждения. *)
(* статус - фильтр промыт. *)
(* подтверждение от фильтра о том, / что он начал промывку. *)
(* импульс о завершении режима промывки фильтра или его аварии. / в последнем фильтре использовать для начала нового цикла. *)
#0 OR(regenerated, filterAlarm, failToRegen)
#1 AND(input, #0)
#2 output <= #1
#3 NOT(#0)
#4 AND(#3, input)
#5 regStatusDelay:TON(IN: startRegen, PT: T#5s)
#6 failureRtrig:R_TRIG(CLK: #5.Q)
#7 NOT(regenFilterStatus)
#8 AND(#6.Q, #7)
#9 failureRS:RS(SET: #8, RESET1: alarmReset)
#10 failToRegen <= #9.Q1
#11 regenFilterOFF:F_TRIG(CLK: regenFilterStatus)
#12 OR(#11.Q, #8)
#13 regStartRS:RS(SET: #4, RESET1: #12)
#14 startRegen <= #13.Q1
#15 OR(#8, #11.Q)
#16 loopFinished <= #15
#17 OR(startNextLoop, failToRegen)
#18 successRS:RS(SET: #11.Q, RESET1: #17)
#19 regenerated <= #18.Q1
_END_CFC_
(* the same logic as Structured Text *)
(* Пока не сброшена ошибка / регенерации, нельзя поставить / отметку, что регенерация прошла. *)
(* запустить новый цикл, сбрасываются все / статусы промытости фильтров, начало / промывок снова от первого фильтра. *)
(* Модуль управления очередью отправок фильтров на промывку. / При поступлении сигнала на промывку от счетчика стоков, подаем сигнал на принудительный перевод в регенерацию на управляющий клапан фильтра. / Принимаем от него сигнал, что он перешел в режим регенерации, подаем сигнал на перевод задвижек этого фильтра в требуемое положение, / если подтверждение не пришло, ставим статус "неудачная попытка регенерации", исключаем этот фильтр из очереди, пока не будет нажат сброс аварии. / Если подтверждение пришло, далее процессом рулит управляющий клапан фильтра. / Он держит сигнал л том, что он в регенерации во время всего процесса промывки. Когда сигнал будет снят, ставим статус, что данный фильтр промыт, / далее будет промываться следующий по очереди фильтр. / Если фильтр, который был в аварии, отремонтирован, нажат сброс аварии, то он будет промыт в следующий сигнал о промывке, вне очереди, или первым / в очереди отремонтированных, после чего пойдет обычная очередь. *)
(* сигнал на запуск промывки. *)
(* если этот фильтр уже промыт, или в аварии, / то передача сигнала на промывку следующему фильтру. / В последнем фильтре не использовать. *)
(* сигнал на начало регенерации / в управляющем клапане фильтра и / перевод задвижек в требуемое состояние: / - если true - промывка; / - если false - фильтрация. *)
(* неудачная попытка запуска регенерации, / от фильтра не поступил сигнал подтверждения. *)
(* статус - фильтр промыт. *)
(* подтверждение от фильтра о том, / что он начал промывку. *)
(* импульс о завершении режима промывки фильтра или его аварии. / в последнем фильтре использовать для начала нового цикла. *)
_t45 := regenerated OR filterAlarm OR failToRegen;
output := input AND _t45;
regStatusDelay(IN := startRegen, PT := T#5s);
failureRtrig(CLK := regStatusDelay.Q);
_t78 := failureRtrig.Q AND NOT regenFilterStatus;
failureRS(SET := _t78, RESET1 := alarmReset);
failToRegen := failureRS.Q1;
regenFilterOFF(CLK := regenFilterStatus);
regStartRS(SET := NOT _t45 AND input, RESET1 := regenFilterOFF.Q OR _t78);
startRegen := regStartRS.Q1;
loopFinished := _t78 OR regenFilterOFF.Q;
successRS(SET := regenFilterOFF.Q, RESET1 := startNextLoop OR failToRegen);
regenerated := successRS.Q1;
END_FUNCTION_BLOCK

(* POU SimpleValve, CFC *)
FUNCTION_BLOCK SimpleValve
VAR_INPUT
	inputOpen: BOOL;			(*вход для подачи импульса на открытие*)
	inputClose: BOOL;		(*вход для подачи импульса на закрытие*)
	statusOpen: BOOL;		(*статус: заслонка/задвижка ОТКРЫТА*)
	statusClose: BOOL;		(*статус: заслонка/задвижка ЗАКРЫТА*)
	reset: BOOL;		(*ручной сброс выходов и аварий в неактивное состояние*)
	timeToOpenClose: WORD;		(*Время в секундах на открытие/закрытие (по тех.характеристикам прибора).*)
END_VAR
VAR_OUTPUT
	outputOpen: BOOL;		(*выход на открытие задвижки/заслонки*)
	outputClose: BOOL;		(*выход на закрытие задвижки/заслонки*)
	errorToOpen: BOOL;		(*авария на открытие - задвижка не открылась за заданное время.*)
	errorToClose: BOOL;		(*авария на закрытие - задвижка не закрылась за заданное время.*)
END_VAR
VAR
	toOpenTrigger: RS;			(*Триггер сигнала на открытие.*)
	toCloseTrigger: RS;			(*Триггер сигнала на закрытие.*)
	timerToOpenClose: TON;		(*Таймер контроля времени открытия/закрытия.*)
	timerToStopOpening: TOF;		(*Задержка на останов открытия заслонки после получения статуса
										открыт от концевиков для плотного закрытия, полного открытия.*)
	timerToStopClosing: TOF;		(*Задержка на останов закрытия заслонки после получения статуса
										закрыт от концевиков для плотного закрытия, полного открытия.*)
	timerToDelayOpen: TOF;		(*Делает паузу 2,5 секунды на открытие после закрытия.*)
	timerToDelayClose: TOF;		(*Делает паузу 2,5 секунды на закрытие после открытия.*)
	statusOpenRS: RS;		(*Защелка сигнала об открытии*)
	statusCloseRS: RS;		(*Защелка сигнала о закрытии*)
END_VAR
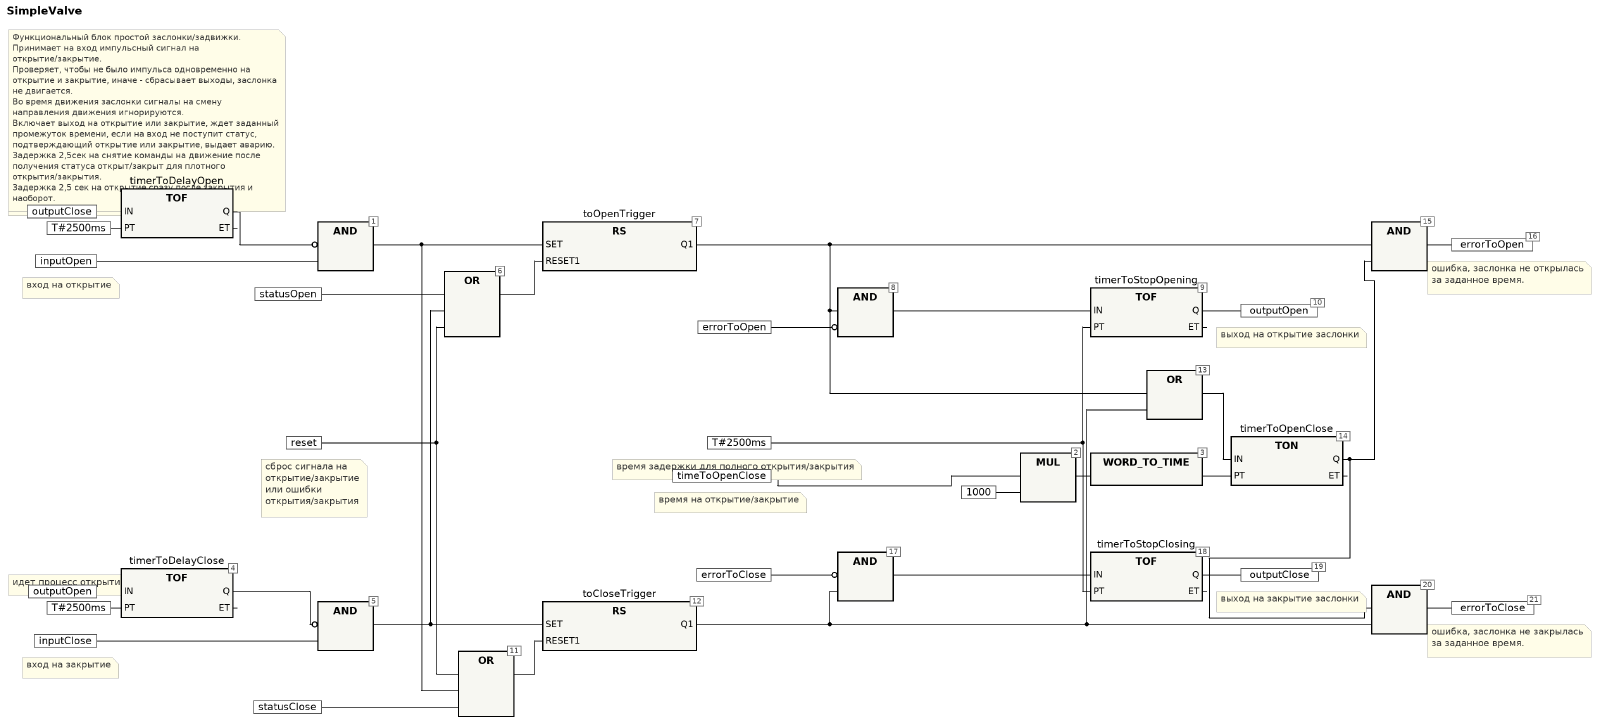
_CFC_ (* Continuous Function Chart, elements in execution order *)
(* идет процесс открытия *)
(* вход на закрытие *)
(* идет процесс закрытия *)
(* сброс сигнала на / открытие/закрытие / или ошибки / открытия/закрытия *)
(* вход на открытие *)
(* Функциональный блок простой заслонки/задвижки. / Принимает на вход импульсный сигнал на открытие/закрытие. / Проверяет, чтобы не было импульса одновременно на открытие и закрытие, иначе - сбрасывает выходы, заслонка не двигается. / Во время движения заслонки сигналы на смену направления движения игнорируются. / Включает выход на открытие или закрытие, ждет заданный промежуток времени, если на вход не поступит статус, подтверждающий открытие или закрытие, выдает аварию. / Задержка 2,5сек на снятие команды на движение после получения статуса открыт/закрыт для плотного открытия/закрытия. / Задержка 2,5 сек на открытие сразу после закрытия и наоборот. *)
(* время задержки для полного открытия/закрытия *)
(* время на открытие/закрытие *)
(* выход на открытие заслонки *)
(* ошибка, заслонка не открылась / за заданное время. *)
(* выход на закрытие заслонки *)
(* ошибка, заслонка не закрылась / за заданное время. *)
#0 timerToDelayOpen:TOF(IN: outputClose, PT: T#2500ms)
#1 AND(NOT #0.Q, inputOpen)
#2 MUL(timeToOpenClose, 1000)
#3 WORD_TO_TIME(#2)
#4 timerToDelayClose:TOF(IN: outputOpen, PT: T#2500ms)
#5 AND(NOT #4.Q, inputClose)
#6 OR(statusOpen, #5, reset)
#7 toOpenTrigger:RS(SET: #1, RESET1: #6)
#8 AND(#7.Q1, NOT errorToOpen)
#9 timerToStopOpening:TOF(IN: #8, PT: T#2500ms)
#10 outputOpen <= #9.Q
#11 OR(reset, #1, statusClose)
#12 toCloseTrigger:RS(SET: #5, RESET1: #11)
#13 OR(#7.Q1, #12.Q1)
#14 timerToOpenClose:TON(IN: #13, PT: #3)
#15 AND(#7.Q1, #14.Q)
#16 errorToOpen <= #15
#17 AND(NOT errorToClose, #12.Q1)
#18 timerToStopClosing:TOF(IN: #17, PT: T#2500ms)
#19 outputClose <= #18.Q
#20 AND(#14.Q, #12.Q1)
#21 errorToClose <= #20
_END_CFC_
END_FUNCTION_BLOCK

(* POU RichTwoPumpManager, CFC *)
FUNCTION_BLOCK RichTwoPumpManager
VAR_INPUT
	start: BOOL;		(*Сигнал на запуск насоса согласно выбранному режиму.*)
	setPump1main: BOOL;		(*Установить режим - насос 1 = главный.
Включать импульсом.*)
	setPump2main: BOOL;		(*Установить режим - насос 2 = главный.
Включать импульсом.*)
	setByCounter: BOOL;		(*Установить режим - по количеству включений.
Включать импульсом.*)
	setByWorkTime: BOOL;		(*Установить режим - по наработке.
Включать импульсом.*)
	resetPump1counter: BOOL;		(*Сброс счетчика количества включений насоса 1.*)
	resetPump2counter: BOOL;		(*Сброс счетчика количества включений насоса 2.*)
	resetWorkTimePump1: BOOL;		(*Сброс счетчика наработки насоса 1.*)
	resetWorkTimePump2: BOOL;		(*Сброс счетчика наработки насоса 2.*)
	startPump1man: BOOL;		(*Пуск насоса 1 вручную независимо от текущего режима.*)
	startPump2man: BOOL;		(*Пуск насоса 2 вручную независимо от текущего режима.*)
	stop: BOOL;		(*Стоп обоих насосов пока вход активен.
Не стоит применять для штатного останова.*)
	resetAlarms: BOOL;		(*Сброс аварий насоса.*)
	delayRepeatedStartTime: WORD;		(*Количество секунд на задержку повторного пуска насоса.
Защита от частых включений. Если ничего не подключено = 300сек.*)
	alarmPump1input: BOOL;		(*Вход от источника сигнала об аварии насоса 1.*)
	alarmPump2input: BOOL;		(*Вход от источника сигнала об аварии насоса 2.*)
END_VAR
VAR_OUTPUT
	regimePump1Main: BOOL;		(*Текущий режим - насос 1 = главный.*)
	regimePump2Main: BOOL;		(*Текущий режим - насос 2 = главный.*)
	regimeByCounter: BOOL;		(*Текущий режим - по количеству включений.*)
	regimeByWorkTime: BOOL;		(*Текущий режим - по наработке.*)
	counterPump1: DWORD;		(*Количество включений насоса 1.*)
	counterPump2: DWORD;		(*Количество включений насоса 2.*)
	daysPump1: WORD;		(*Количество отработанных дней насоса 1.*)
	hoursPump1: WORD;		(*Количество отработанных часов насоса 1.*)
	minutesPump1: WORD;		(*Количество отработанных минут насоса 1.*)
	secondsPump1: WORD;		(*Количество отработанных секунд насоса 1.*)
	daysPump2: WORD;		(*Количество отработанных дней насоса 2.*)
	hoursPump2: WORD;		(*Количество отработанных часов насоса 2.*)
	minutesPump2: WORD;		(*Количество отработанных минут насоса 2.*)
	secondsPump2: WORD;		(*Количество отработанных секунд насоса 2.*)
	pump1starter: BOOL;		(*Сигнал на запуск насоса 1.*)
	pump2starter: BOOL;		(*Сигнал на запуск насоса 2.*)
	nextStartP1timer: WORD;		(*Обратный отсчет до возможности повторного пуска насоса 1.*)
	nextStartP2timer: WORD;		(*Обратный отсчет до возможности повторного пуска насоса 2.*)
	alarmPump1output: BOOL;		(*Сигнал авария насоса 1.
Триггерится, нужен сброс.*)
	alarmPump2output: BOOL;		(*Сигнал авария насоса 2.
Триггерится, нужен сброс.*)
END_VAR
VAR
	ChoosePumpRegime: ChoosePumpRegime;		(*Блок выбора режима включения.*)
	CounterManager: CounterManager;		(*Блок выбора и запуска насоса по наработке.*)
	WorkTimeManager: WorkTimeManager;		(*Блок выбора и запуска насоса с меньшей наработкой.*)
	simpleTimeManager: SimpleTwoPumpManager;		(*Блок управления двумя насосами, горячий резерв, автоматическое переключение.*)
END_VAR
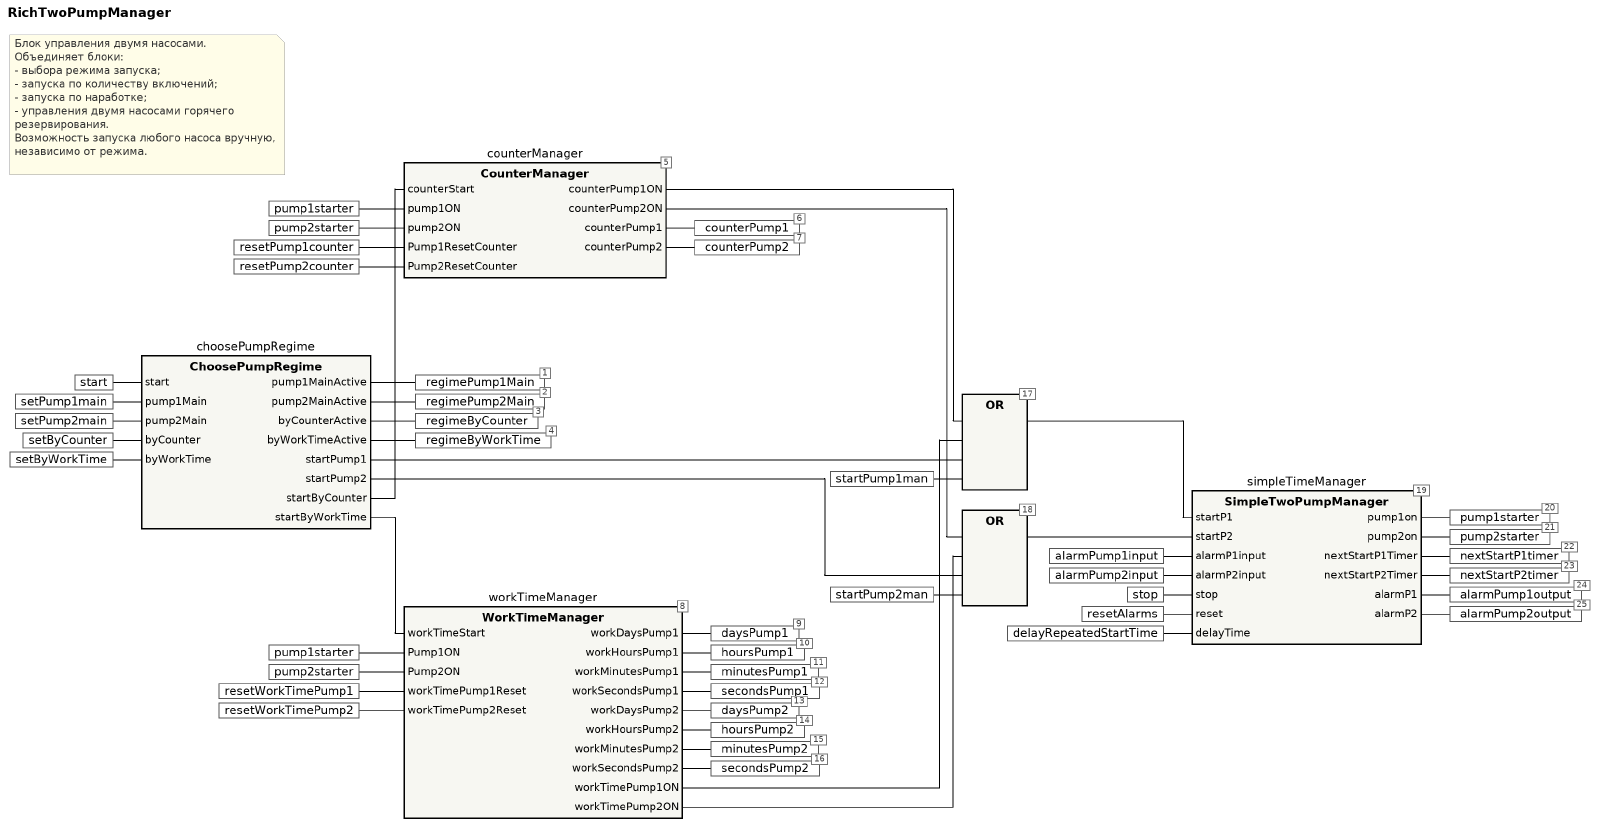
_CFC_ (* Continuous Function Chart, elements in execution order *)
(* Блок управления двумя насосами. / Объединяет блоки: / - выбора режима запуска; / - запуска по количеству включений; / - запуска по наработке; / - управления двумя насосами горячего резервирования. / Возможность запуска любого насоса вручную, / независимо от режима. *)
#0 choosePumpRegime:ChoosePumpRegime(start: start, pump1Main: setPump1main, pump2Main: setPump2main, byCounter: setByCounter, byWorkTime: setByWorkTime)
#1 regimePump1Main <= #0.pump1MainActive
#2 regimePump2Main <= #0.pump2MainActive
#3 regimeByCounter <= #0.byCounterActive
#4 regimeByWorkTime <= #0.byWorkTimeActive
#5 counterManager:CounterManager(counterStart: #0.startByCounter, pump1ON: pump1starter, pump2ON: pump2starter, Pump1ResetCounter: resetPump1counter, Pump2ResetCounter: resetPump2counter)
#6 counterPump1 <= #5.counterPump1
#7 counterPump2 <= #5.counterPump2
#8 workTimeManager:WorkTimeManager(workTimeStart: #0.startByWorkTime, Pump1ON: pump1starter, Pump2ON: pump2starter, workTimePump1Reset: resetWorkTimePump1, workTimePump2Reset: resetWorkTimePump2)
#9 daysPump1 <= #8.workDaysPump1
#10 hoursPump1 <= #8.workHoursPump1
#11 minutesPump1 <= #8.workMinutesPump1
#12 secondsPump1 <= #8.workSecondsPump1
#13 daysPump2 <= #8.workDaysPump2
#14 hoursPump2 <= #8.workHoursPump2
#15 minutesPump2 <= #8.workMinutesPump2
#16 secondsPump2 <= #8.workSecondsPump2
#17 OR(#5.counterPump1ON, #8.workTimePump1ON, #0.startPump1, startPump1man)
#18 OR(#5.counterPump2ON, #8.workTimePump2ON, #0.startPump2, startPump2man)
#19 simpleTimeManager:SimpleTwoPumpManager(startP1: #17, startP2: #18, alarmP1input: alarmPump1input, alarmP2input: alarmPump2input, stop: stop, reset: resetAlarms, delayTime: delayRepeatedStartTime)
#20 pump1starter <= #19.pump1on
#21 pump2starter <= #19.pump2on
#22 nextStartP1timer <= #19.nextStartP1Timer
#23 nextStartP2timer <= #19.nextStartP2Timer
#24 alarmPump1output <= #19.alarmP1
#25 alarmPump2output <= #19.alarmP2
_END_CFC_
(* the same logic as Structured Text *)
(* Блок управления двумя насосами. / Объединяет блоки: / - выбора режима запуска; / - запуска по количеству включений; / - запуска по наработке; / - управления двумя насосами горячего резервирования. / Возможность запуска любого насоса вручную, / независимо от режима. *)
choosePumpRegime(start := start, pump1Main := setPump1main, pump2Main := setPump2main, byCounter := setByCounter, byWorkTime := setByWorkTime);
regimePump1Main := choosePumpRegime.pump1MainActive;
regimePump2Main := choosePumpRegime.pump2MainActive;
regimeByCounter := choosePumpRegime.byCounterActive;
regimeByWorkTime := choosePumpRegime.byWorkTimeActive;
counterManager(counterStart := choosePumpRegime.startByCounter, pump1ON := pump1starter, pump2ON := pump2starter, Pump1ResetCounter := resetPump1counter, Pump2ResetCounter := resetPump2counter);
counterPump1 := counterManager.counterPump1;
counterPump2 := counterManager.counterPump2;
workTimeManager(workTimeStart := choosePumpRegime.startByWorkTime, Pump1ON := pump1starter, Pump2ON := pump2starter, workTimePump1Reset := resetWorkTimePump1, workTimePump2Reset := resetWorkTimePump2);
daysPump1 := workTimeManager.workDaysPump1;
hoursPump1 := workTimeManager.workHoursPump1;
minutesPump1 := workTimeManager.workMinutesPump1;
secondsPump1 := workTimeManager.workSecondsPump1;
daysPump2 := workTimeManager.workDaysPump2;
hoursPump2 := workTimeManager.workHoursPump2;
minutesPump2 := workTimeManager.workMinutesPump2;
secondsPump2 := workTimeManager.workSecondsPump2;
simpleTimeManager(startP1 := counterManager.counterPump1ON OR workTimeManager.workTimePump1ON OR choosePumpRegime.startPump1 OR startPump1man, startP2 := counterManager.counterPump2ON OR workTimeManager.workTimePump2ON OR choosePumpRegime.startPump2 OR startPump2man, alarmP1input := alarmPump1input, alarmP2input := alarmPump2input, stop := stop, reset := resetAlarms, delayTime := delayRepeatedStartTime);
pump1starter := simpleTimeManager.pump1on;
pump2starter := simpleTimeManager.pump2on;
nextStartP1timer := simpleTimeManager.nextStartP1Timer;
nextStartP2timer := simpleTimeManager.nextStartP2Timer;
alarmPump1output := simpleTimeManager.alarmP1;
alarmPump2output := simpleTimeManager.alarmP2;
END_FUNCTION_BLOCK

(* POU WorkTimeManager, CFC *)
FUNCTION_BLOCK WorkTimeManager
VAR
	workTimePump1: TimeSeparator;		(*Блок вывода времени наработки  насоса 1.*)
	workTimePump2: TimeSeparator;		(*Блок вывода времени наработки насоса 2.*)
	currentWorkTimePump1: DWORD;		(*Текущая наработка в секундах насоса 1.*)
	currentWorkTimePump2: DWORD;		(*Текущая наработка в секундах насоса 2.*)
	pulsarP1: PulsePerSec;		(*Генератор импульса в секунду для наработки насоса 1.*)
	pulsarP2: PulsePerSec;		(*Генератор импульса в секунду для наработки насоса 2.*)
	timeStartRtrig: R_TRIG;		(*Детектор переднего фронта сигнала на запуск.*)
	timeStartFtrig: F_TRIG;		(*Детектор спада сигнала на запуск.*)
	RStrigTimePump1: RS;		(*RSтриггер сигнала на запуск насоса 1.*)
	RStrigTimePump2: RS;		(*RSтриггер сигнала на запуск насоса 2.*)
END_VAR
VAR_OUTPUT
	workDaysPump1: WORD;		(*Количество отработанных дней для насоса 1.*)
	workHoursPump1: WORD;		(*Количество отработанных часов для насоса 1.*)
	workMinutesPump1: WORD;		(*Количество отработанных минут для насоса 1.*)
	workSecondsPump1: WORD;		(*Количество отработанных секунд для насоса 1.*)
	workDaysPump2: WORD;		(*Количество отработанных дней для насоса 2.*)
	workHoursPump2: WORD;		(*Количество отработанных часов для насоса 2.*)
	workMinutesPump2: WORD;		(*Количество отработанных минут для насоса 2.*)
	workSecondsPump2: WORD;		(*Количество отработанных секунд для насоса 2.*)
	workTimePump1ON: BOOL;		(*Выход на запуск насоса 1.*)
	workTimePump2ON: BOOL;		(*Выход на запуск насоса 2.*)
END_VAR
VAR_INPUT
	workTimeStart: BOOL;		(*Сигнал на запуск насоса с наименьшим временем работы.*)
	Pump1ON: BOOL;		(*Сигнал подтверждение о запуске насоса 1.*)
	Pump2ON: BOOL;		(*Сигнал подтверждение о запуске насоса 2.*)
	workTimePump1Reset: BOOL;		(*Сброс времени наработки насоса 1.*)
	workTimePump2Reset: BOOL;		(*Сброс времени наработки насоса 2.*)
END_VAR
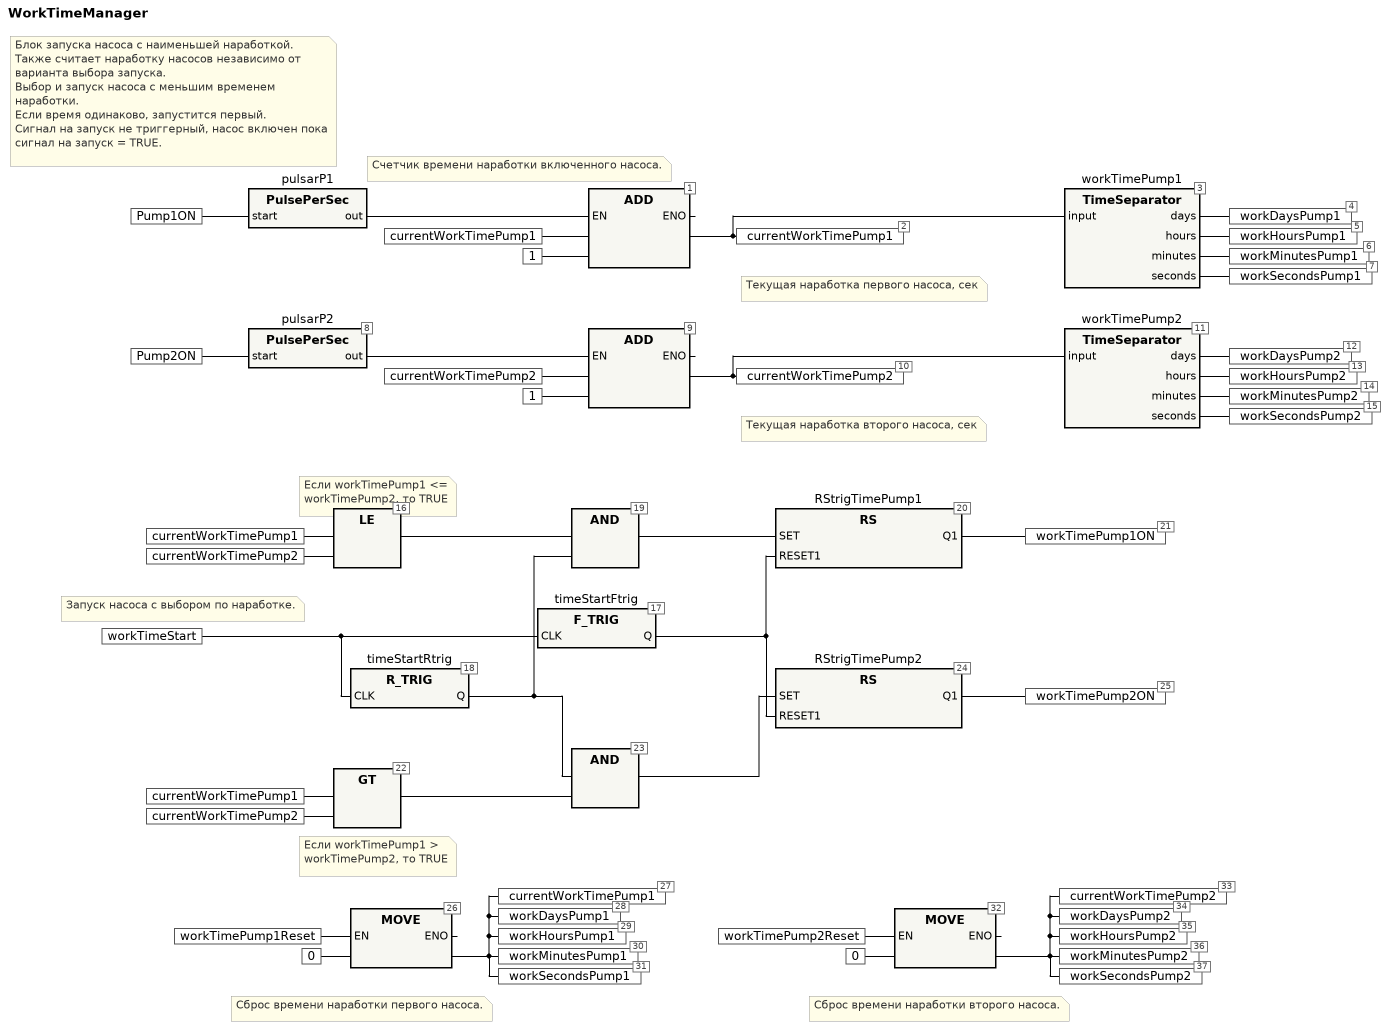
_CFC_ (* Continuous Function Chart, elements in execution order *)
(* Текущая наработка второго насоса, сек *)
(* Сброс времени наработки второго насоса. *)
(* Текущая наработка первого насоса, сек *)
(* Счетчик времени наработки включенного насоса. *)
(* Если workTimePump1 > / workTimePump2, то TRUE *)
(* Если workTimePump1 <= / workTimePump2, то TRUE *)
(* Запуск насоса с выбором по наработке. *)
(* Блок запуска насоса с наименьшей наработкой. / Также считает наработку насосов независимо от варианта выбора запуска. / Выбор и запуск насоса с меньшим временем наработки. / Если время одинаково, запустится первый. / Сигнал на запуск не триггерный, насос включен пока сигнал на запуск = TRUE. *)
(* Сброс времени наработки первого насоса. *)
#0 pulsarP1:PulsePerSec(start: Pump1ON)
#1 ADD(EN: #0.out, currentWorkTimePump1, 1)
#2 currentWorkTimePump1 <= #1
#3 workTimePump1:TimeSeparator(input: #1)
#4 workDaysPump1 <= #3.days
#5 workHoursPump1 <= #3.hours
#6 workMinutesPump1 <= #3.minutes
#7 workSecondsPump1 <= #3.seconds
#8 pulsarP2:PulsePerSec(start: Pump2ON)
#9 ADD(EN: #8.out, currentWorkTimePump2, 1)
#10 currentWorkTimePump2 <= #9
#11 workTimePump2:TimeSeparator(input: #9)
#12 workDaysPump2 <= #11.days
#13 workHoursPump2 <= #11.hours
#14 workMinutesPump2 <= #11.minutes
#15 workSecondsPump2 <= #11.seconds
#16 LE(currentWorkTimePump1, currentWorkTimePump2)
#17 timeStartFtrig:F_TRIG(CLK: workTimeStart)
#18 timeStartRtrig:R_TRIG(CLK: workTimeStart)
#19 AND(#16, #18.Q)
#20 RStrigTimePump1:RS(SET: #19, RESET1: #17.Q)
#21 workTimePump1ON <= #20.Q1
#22 GT(currentWorkTimePump1, currentWorkTimePump2)
#23 AND(#18.Q, #22)
#24 RStrigTimePump2:RS(SET: #23, RESET1: #17.Q)
#25 workTimePump2ON <= #24.Q1
#26 MOVE(EN: workTimePump1Reset, 0)
#27 currentWorkTimePump1 <= #26
#28 workDaysPump1 <= #26
#29 workHoursPump1 <= #26
#30 workMinutesPump1 <= #26
#31 workSecondsPump1 <= #26
#32 MOVE(EN: workTimePump2Reset, 0)
#33 currentWorkTimePump2 <= #32
#34 workDaysPump2 <= #32
#35 workHoursPump2 <= #32
#36 workMinutesPump2 <= #32
#37 workSecondsPump2 <= #32
_END_CFC_
END_FUNCTION_BLOCK

(* POU TimeSeparator, ST *)
FUNCTION_BLOCK TimeSeparator
VAR_INPUT
	 input: DWORD; (*Вход счетчика  наработки и т.п., сек.*)
END_VAR
VAR_OUTPUT
	days: WORD; (*Выход наработка, дней*)
	hours: WORD; (*Выход наработка, часов*)
	minutes: WORD; (*Выход наработка, минут*)
	seconds: WORD; (*Выход наработка, секунд*)
END_VAR
VAR
	temp: DWORD;
END_VAR
days:= DWORD_TO_WORD (input / (60 * 60 * 24));
temp:= input MOD (60 * 60 * 24);
hours:= DWORD_TO_WORD (temp / (60 * 60));
temp:= temp MOD (60 * 60);
minutes:= DWORD_TO_WORD (temp / 60);
temp:= temp MOD 60;
seconds:= DWORD_TO_WORD (temp);
END_FUNCTION_BLOCK

(* POU SimpleTwoPumpManager, CFC *)
FUNCTION_BLOCK SimpleTwoPumpManager

VAR
	alarmP1trig: RS;		(*Триггер - защелка аварии насоса 1.*)
	alarmP2trig: RS;		(*Триггер - защелка аварии насоса 2.*)
	stopPump1Detector: F_TRIG;		(*Детектор спада сигнала (останов) насоса 1.*)
	stopPump2Detector: F_TRIG;		(*Детектор спада сигнала (останов) насоса 2.*)
	delayAfterStopP2: TOF;		(*Таймер задержки на включение
насоса 1 после останова насоса 2.*)
	delayAfterStopP1: TOF;		(*Таймер задержки на включение
насоса 2 после останова насоса 1.*)
	antiFreqStartPump1: TOF;		(*Таймер - предохранитель от частых пусков насоса 1.*)
	antiFreqStartPump2: TOF;		(*Таймер - предохранитель от частых пусков насоса 2.*)
	startPump1Trig: RS;		(*RS триггер на пуск насоса 1.*)
	startPump2Trig: RS;		(*RS триггер на пуск насоса 2.*)
	stopPump1: F_TRIG;		(*Сигнал на останов насоса 1.*)
	stopPump2: F_TRIG;		(*Сигнал на останов насоса 2.*)
END_VAR
VAR_INPUT
	startP1: BOOL;		(*Сигнал на запуск насоса 1.
Активен - пуск, неактивен - стоп.*)
	startP2: BOOL;		(*Сигнал на запуск насоса 2.
Активен - пуск, неактивен - стоп.*)
	alarmP1input: BOOL;		(*Сигнал авария от насоса 1.*)
	alarmP2input: BOOL;		(*Сигнал авария от насоса 2.*)
	stop: BOOL;		(*Сигнал на останов. Пока активен - пусков нет.
Общий на оба насоса.*)
	reset: BOOL;		(*Сброс аварий.*)
	delayTime: WORD := 300;		(*Задержка на повторный пуск в секундах.
Если ко входу ничего не подключено, то 300сек.*)
END_VAR
VAR_OUTPUT
	pump1on: BOOL;		(*Выход на запуск насоса 1.*)
	pump2on: BOOL;		(*Выход на запуск насоса 2.*)
	nextStartP1Timer: WORD;		(*Счетчик секунд до возможности повторного пуска насоса 1.*)
	nextStartP2Timer: WORD;		(*Счетчик секунд до возможности повторного пуска насоса 2.*)
	alarmP1: BOOL;		(*Статус - авария насоса 1.*)
	alarmP2: BOOL;		(*Статус - авария насоса 2.*)
END_VAR
VAR (* helpers for the ST form of the networks *)
	_t203 : TIME;
END_VAR
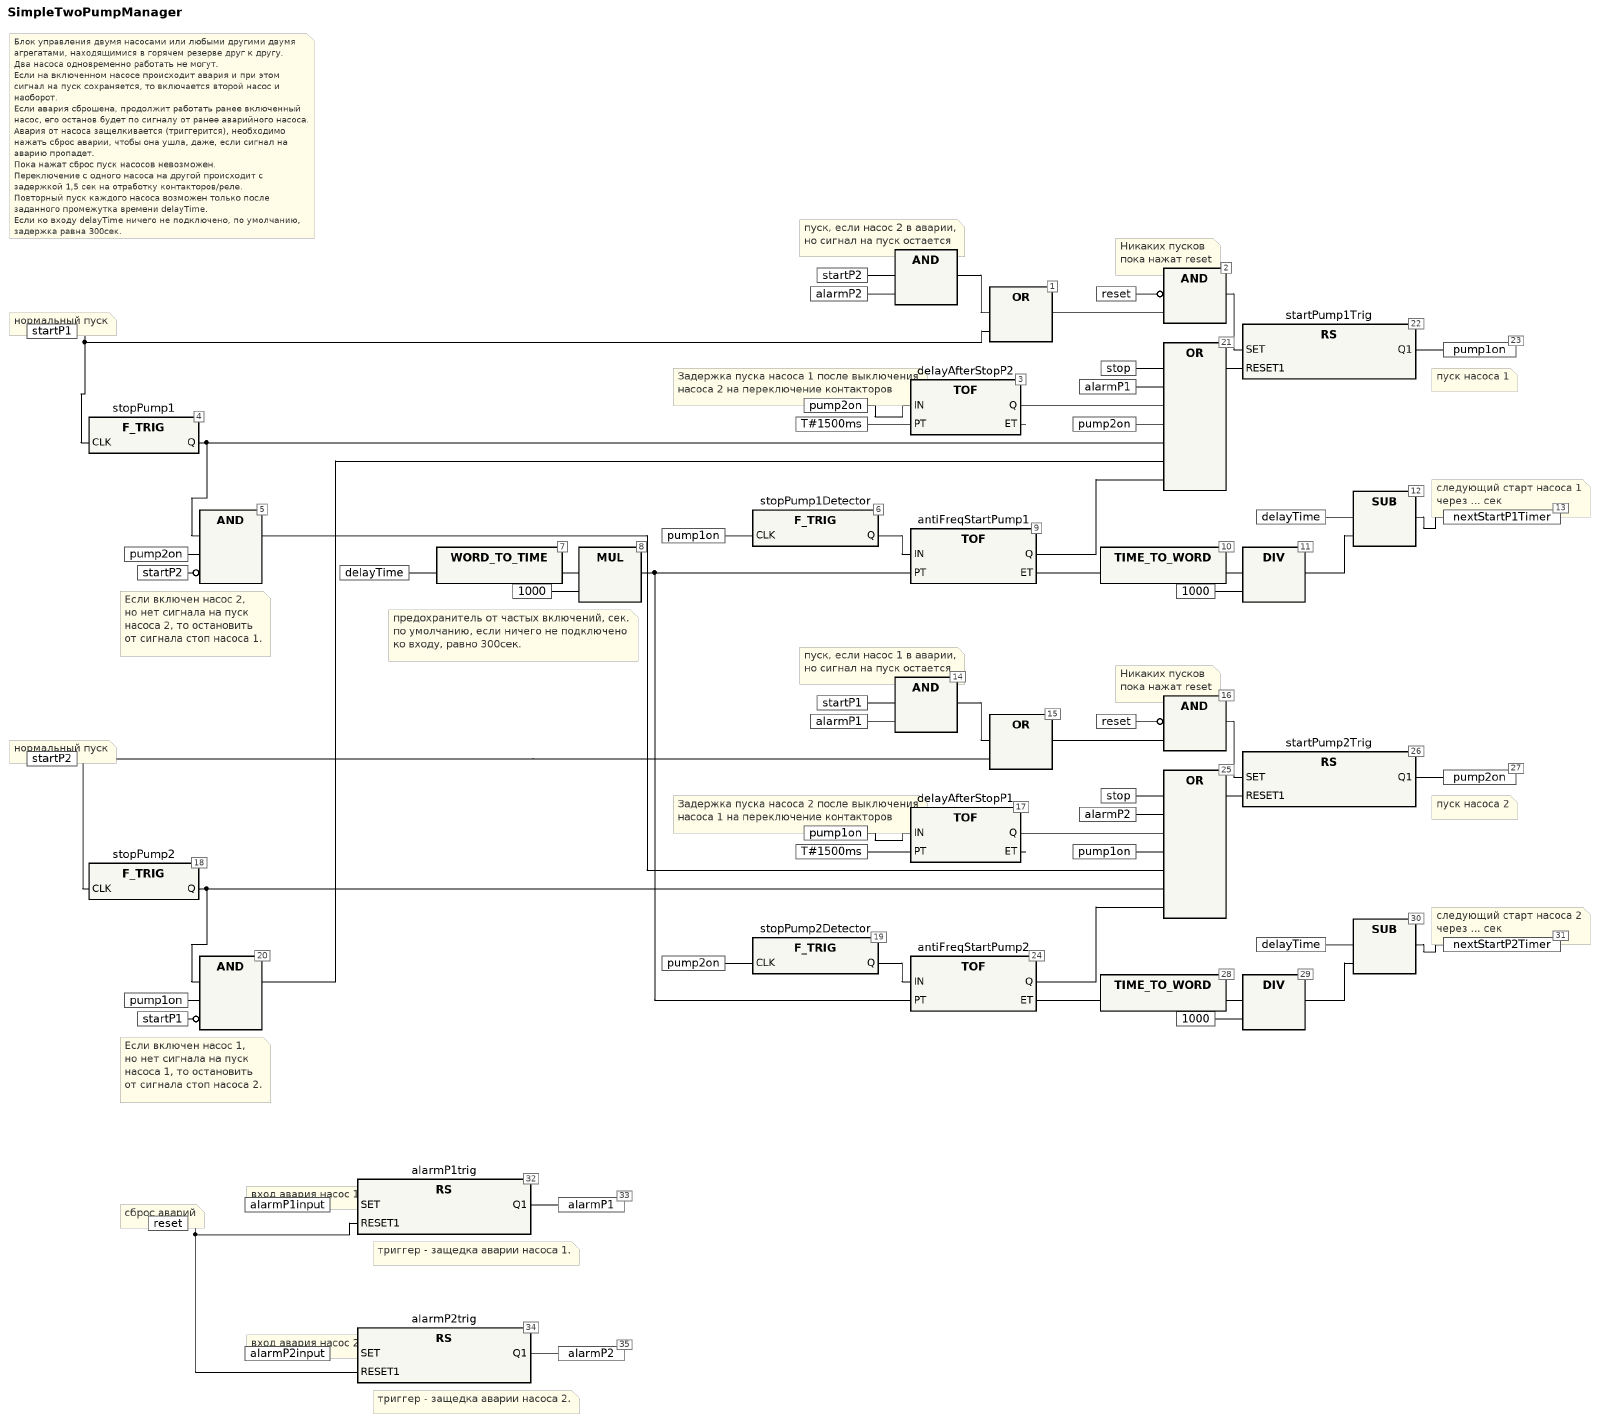
_CFC_ (* Continuous Function Chart, elements in execution order *)
(* Задержка пуска насоса 2 после выключения / насоса 1 на переключение контакторов *)
(* cледующий старт насоса 2 / через ... сек *)
(* триггер - защедка аварии насоса 2. *)
(* cледующий старт насоса 1 / через ... сек *)
(* триггер - защедка аварии насоса 1. *)
(* предохранитель от частых включений, сек. / по умолчанию, если ничего не подключено / ко входу, равно 300сек. *)
(* пуск, если насос 1 в аварии, / но сигнал на пуск остается *)
(* нормальный пуск *)
(* пуск, если насос 2 в аварии, / но сигнал на пуск остается *)
(* нормальный пуск *)
(* Задержка пуска насоса 1 после выключения / насоса 2 на переключение контакторов *)
(* вход авария насос 1 *)
(* сброс аварий *)
(* пуск насоса 1 *)
(* вход авария насос 2 *)
(* пуск насоса 2 *)
(* Блок управления двумя насосами или любыми другими двумя агрегатами, находящимися в горячем резерве друг к другу. / Два насоса одновременно работать не могут. / Если на включенном насосе происходит авария и при этом сигнал на пуск сохраняется, то включается второй насос и наоборот. / Если авария сброшена, продолжит работать ранее включенный насос, его останов будет по сигналу от ранее аварийного насоса. / Авария от насоса защелкивается (триггерится), необходимо нажать сброс аварии, чтобы она ушла, даже, если сигнал на аварию пропадет. / Пока нажат сброс пуск насосов невозможен. / Переключение с одного насоса на другой происходит с задержкой 1,5 сек на отработку контакторов/реле. / Повторный пуск каждого насоса возможен только после заданного промежутка времени delayTime. / Если ко входу delayTime ничего не подключено, по умолчанию, задержка равна 300сек. *)
(* Никаких пусков / пока нажат reset *)
(* Никаких пусков / пока нажат reset *)
(* Если включен насос 2, / но нет сигнала на пуск / насоса 2, то остановить / от сигнала стоп насоса 1. *)
(* Если включен насос 1, / но нет сигнала на пуск / насоса 1, то остановить / от сигнала стоп насоса 2. *)
#0 AND(startP2, alarmP2)
#1 OR(#0, startP1)
#2 AND(NOT reset, #1)
#3 delayAfterStopP2:TOF(IN: pump2on, PT: T#1500ms)
#4 stopPump1:F_TRIG(CLK: startP1)
#5 AND(#4.Q, pump2on, NOT startP2)
#6 stopPump1Detector:F_TRIG(CLK: pump1on)
#7 WORD_TO_TIME(delayTime)
#8 MUL(#7, 1000)
#9 antiFreqStartPump1:TOF(IN: #6.Q, PT: #8)
#10 TIME_TO_WORD(#9.ET)
#11 DIV(#10, 1000)
#12 SUB(delayTime, #11)
#13 nextStartP1Timer <= #12
#14 AND(startP1, alarmP1)
#15 OR(#14, startP2)
#16 AND(NOT reset, #15)
#17 delayAfterStopP1:TOF(IN: pump1on, PT: T#1500ms)
#18 stopPump2:F_TRIG(CLK: startP2)
#19 stopPump2Detector:F_TRIG(CLK: pump2on)
#20 AND(#18.Q, pump1on, NOT startP1)
#21 OR(stop, alarmP1, #3.Q, pump2on, #4.Q, #20, #9.Q)
#22 startPump1Trig:RS(SET: #2, RESET1: #21)
#23 pump1on <= #22.Q1
#24 antiFreqStartPump2:TOF(IN: #19.Q, PT: #8)
#25 OR(stop, alarmP2, #17.Q, pump1on, #5, #18.Q, #24.Q)
#26 startPump2Trig:RS(SET: #16, RESET1: #25)
#27 pump2on <= #26.Q1
#28 TIME_TO_WORD(#24.ET)
#29 DIV(#28, 1000)
#30 SUB(delayTime, #29)
#31 nextStartP2Timer <= #30
#32 alarmP1trig:RS(SET: alarmP1input, RESET1: reset)
#33 alarmP1 <= #32.Q1
#34 alarmP2trig:RS(SET: alarmP2input, RESET1: reset)
#35 alarmP2 <= #34.Q1
_END_CFC_
(* the same logic as Structured Text *)
(* Задержка пуска насоса 2 после выключения / насоса 1 на переключение контакторов *)
(* cледующий старт насоса 2 / через ... сек *)
(* триггер - защедка аварии насоса 2. *)
(* cледующий старт насоса 1 / через ... сек *)
(* триггер - защедка аварии насоса 1. *)
(* предохранитель от частых включений, сек. / по умолчанию, если ничего не подключено / ко входу, равно 300сек. *)
(* пуск, если насос 1 в аварии, / но сигнал на пуск остается *)
(* нормальный пуск *)
(* пуск, если насос 2 в аварии, / но сигнал на пуск остается *)
(* нормальный пуск *)
(* Задержка пуска насоса 1 после выключения / насоса 2 на переключение контакторов *)
(* вход авария насос 1 *)
(* сброс аварий *)
(* пуск насоса 1 *)
(* вход авария насос 2 *)
(* пуск насоса 2 *)
(* Блок управления двумя насосами или любыми другими двумя агрегатами, находящимися в горячем резерве друг к другу. / Два насоса одновременно работать не могут. / Если на включенном насосе происходит авария и при этом сигнал на пуск сохраняется, то включается второй насос и наоборот. / Если авария сброшена, продолжит работать ранее включенный насос, его останов будет по сигналу от ранее аварийного насоса. / Авария от насоса защелкивается (триггерится), необходимо нажать сброс аварии, чтобы она ушла, даже, если сигнал на аварию пропадет. / Пока нажат сброс пуск насосов невозможен. / Переключение с одного насоса на другой происходит с задержкой 1,5 сек на отработку контакторов/реле. / Повторный пуск каждого насоса возможен только после заданного промежутка времени delayTime. / Если ко входу delayTime ничего не подключено, по умолчанию, задержка равна 300сек. *)
(* Никаких пусков / пока нажат reset *)
(* Никаких пусков / пока нажат reset *)
(* Если включен насос 2, / но нет сигнала на пуск / насоса 2, то остановить / от сигнала стоп насоса 1. *)
(* Если включен насос 1, / но нет сигнала на пуск / насоса 1, то остановить / от сигнала стоп насоса 2. *)
delayAfterStopP2(IN := pump2on, PT := T#1500ms);
stopPump1(CLK := startP1);
stopPump1Detector(CLK := pump1on);
_t203 := WORD_TO_TIME(delayTime) * 1000;
antiFreqStartPump1(IN := stopPump1Detector.Q, PT := _t203);
nextStartP1Timer := delayTime - (TIME_TO_WORD(antiFreqStartPump1.ET) / 1000);
delayAfterStopP1(IN := pump1on, PT := T#1500ms);
stopPump2(CLK := startP2);
stopPump2Detector(CLK := pump2on);
startPump1Trig(SET := NOT reset AND ((startP2 AND alarmP2) OR startP1), RESET1 := stop OR alarmP1 OR delayAfterStopP2.Q OR pump2on OR stopPump1.Q OR (stopPump2.Q AND pump1on AND NOT startP1) OR antiFreqStartPump1.Q);
pump1on := startPump1Trig.Q1;
antiFreqStartPump2(IN := stopPump2Detector.Q, PT := _t203);
startPump2Trig(SET := NOT reset AND ((startP1 AND alarmP1) OR startP2), RESET1 := stop OR alarmP2 OR delayAfterStopP1.Q OR pump1on OR (stopPump1.Q AND pump2on AND NOT startP2) OR stopPump2.Q OR antiFreqStartPump2.Q);
pump2on := startPump2Trig.Q1;
nextStartP2Timer := delayTime - (TIME_TO_WORD(antiFreqStartPump2.ET) / 1000);
alarmP1trig(SET := alarmP1input, RESET1 := reset);
alarmP1 := alarmP1trig.Q1;
alarmP2trig(SET := alarmP2input, RESET1 := reset);
alarmP2 := alarmP2trig.Q1;
END_FUNCTION_BLOCK

(* POU TwoPumpOneDriveManager, CFC *)
FUNCTION_BLOCK TwoPumpOneDriveManager
	VAR_INPUT
	start: BOOL;		(*Сигнал на запуск насоса согласно выбранному режиму.*)
	setPump1main: BOOL;		(*Установить режим - насос 1 = главный.
Включать импульсом.*)
	setPump2main: BOOL;		(*Установить режим - насос 2 = главный.
Включать импульсом.*)
	setByCounter: BOOL;		(*Установить режим - по количеству включений.
Включать импульсом.*)
	setByWorkTime: BOOL;		(*Установить режим - по наработке.
Включать импульсом.*)
	resetPump1counter: BOOL;		(*Сброс счетчика количества включений насоса 1.*)
	resetPump2counter: BOOL;		(*Сброс счетчика количества включений насоса 2.*)
	resetWorkTimePump1: BOOL;		(*Сброс счетчика наработки насоса 1.*)
	resetWorkTimePump2: BOOL;		(*Сброс счетчика наработки насоса 2.*)
	startPump1man: BOOL;		(*Пуск насоса 1 вручную независимо от текущего режима.*)
	startPump2man: BOOL;		(*Пуск насоса 2 вручную независимо от текущего режима.*)
	stop: BOOL;		(*Стоп обоих насосов пока вход активен.
Не стоит применять для штатного останова.*)
	resetAlarms: BOOL;		(*Сброс аварий насоса.*)
	delayRepeatedStartTime: WORD;		(*Количество секунд на задержку повторного пуска насоса.
Защита от частых включений. Если ничего не подключено = 300сек.*)
	alarmPump1input: BOOL;		(*Вход от источника сигнала об аварии насоса 1.*)
	alarmPump2input: BOOL;		(*Вход от источника сигнала об аварии насоса 2.*)
	driveAlarm: BOOL;		(*Сигнал авария от ЧРП.*)
END_VAR
VAR_OUTPUT
	regimePump1Main: BOOL;		(*Текущий режим - насос 1 = главный.*)
	regimePump2Main: BOOL;		(*Текущий режим - насос 2 = главный.*)
	regimeByCounter: BOOL;		(*Текущий режим - по количеству включений.*)
	regimeByWorkTime: BOOL;		(*Текущий режим - по наработке.*)
	counterPump1: DWORD;		(*Количество включений насоса 1.*)
	counterPump2: DWORD;		(*Количество включений насоса 2.*)
	daysPump1: WORD;		(*Количество отработанных дней насоса 1.*)
	hoursPump1: WORD;		(*Количество отработанных часов насоса 1.*)
	minutesPump1: WORD;		(*Количество отработанных минут насоса 1.*)
	secondsPump1: WORD;		(*Количество отработанных секунд насоса 1.*)
	daysPump2: WORD;		(*Количество отработанных дней насоса 2.*)
	hoursPump2: WORD;		(*Количество отработанных часов насоса 2.*)
	minutesPump2: WORD;		(*Количество отработанных минут насоса 2.*)
	secondsPump2: WORD;		(*Количество отработанных секунд насоса 2.*)
	drivePower: BOOL;		(*Сигнал на включение контактора частотного преобразователя.*)
	pump1ON: BOOL;		(*Сигнал на включение контактора насоса 1.*)
	pump2ON: BOOL;		(*Сигнал на включение контактора насоса 2.*)
	startDrive: BOOL;		(*Сигнал на запуск в частотный преобразователь.*)
	nextStartP1timer: WORD;		(*Обратный отсчет до возможности повторного пуска насоса 1.*)
	nextStartP2timer: WORD;		(*Обратный отсчет до возможности повторного пуска насоса 2.*)
	alarmPump1output: BOOL;		(*Сигнал авария насоса 1.
Триггерится, нужен сброс.*)
	alarmPump2output: BOOL;		(*Сигнал авария насоса 2.
Триггерится, нужен сброс.*)
END_VAR
VAR

	RichTwoPumpManager: RichTwoPumpManager;		(*Блок управления двумя насосами.*)
	TwoPumpOneDriveModule: TwoPumpOneDriveModule;		(*Модуль управления контакторами двух насосов и питания одного частотного преобразователя.*)
END_VAR
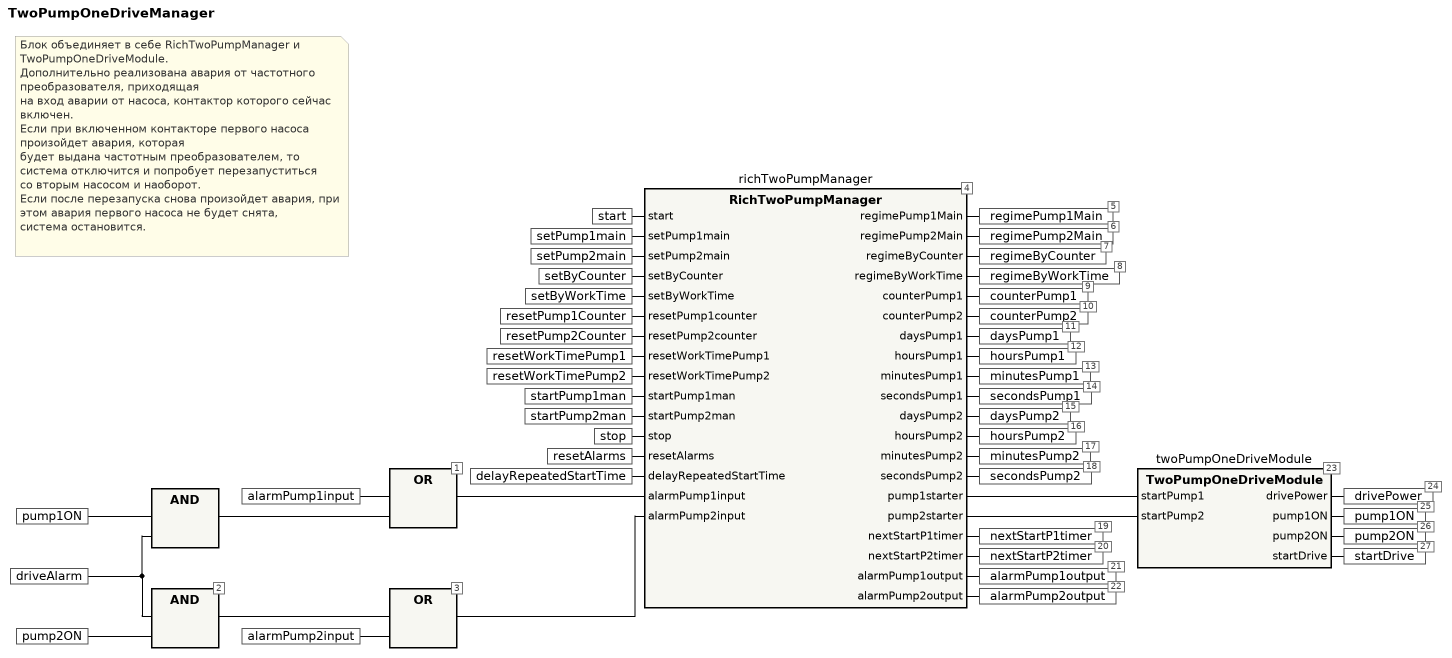
_CFC_ (* Continuous Function Chart, elements in execution order *)
(* Блок объединяет в себе RichTwoPumpManager и TwoPumpOneDriveModule. / Дополнительно реализована авария от частотного преобразователя, приходящая / на вход аварии от насоса, контактор которого сейчас включен. / Если при включенном контакторе первого насоса произойдет авария, которая / будет выдана частотным преобразователем, то система отключится и попробует перезапуститься / со вторым насосом и наоборот. / Если после перезапуска снова произойдет авария, при этом авария первого насоса не будет снята, / система остановится. *)
#0 AND(pump1ON, driveAlarm)
#1 OR(alarmPump1input, #0)
#2 AND(driveAlarm, pump2ON)
#3 OR(#2, alarmPump2input)
#4 richTwoPumpManager:RichTwoPumpManager(start: start, setPump1main: setPump1main, setPump2main: setPump2main, setByCounter: setByCounter, setByWorkTime: setByWorkTime, resetPump1counter: resetPump1Counter, resetPump2counter: resetPump2Counter, resetWorkTimePump1: resetWorkTimePump1, resetWorkTimePump2: resetWorkTimePump2, startPump1man: startPump1man, startPump2man: startPump2man, stop: stop, resetAlarms: resetAlarms, delayRepeatedStartTime: delayRepeatedStartTime, alarmPump1input: #1, alarmPump2input: #3)
#5 regimePump1Main <= #4.regimePump1Main
#6 regimePump2Main <= #4.regimePump2Main
#7 regimeByCounter <= #4.regimeByCounter
#8 regimeByWorkTime <= #4.regimeByWorkTime
#9 counterPump1 <= #4.counterPump1
#10 counterPump2 <= #4.counterPump2
#11 daysPump1 <= #4.daysPump1
#12 hoursPump1 <= #4.hoursPump1
#13 minutesPump1 <= #4.minutesPump1
#14 secondsPump1 <= #4.secondsPump1
#15 daysPump2 <= #4.daysPump2
#16 hoursPump2 <= #4.hoursPump2
#17 minutesPump2 <= #4.minutesPump2
#18 secondsPump2 <= #4.secondsPump2
#19 nextStartP1timer <= #4.nextStartP1timer
#20 nextStartP2timer <= #4.nextStartP2timer
#21 alarmPump1output <= #4.alarmPump1output
#22 alarmPump2output <= #4.alarmPump2output
#23 twoPumpOneDriveModule:TwoPumpOneDriveModule(startPump1: #4.pump1starter, startPump2: #4.pump2starter)
#24 drivePower <= #23.drivePower
#25 pump1ON <= #23.pump1ON
#26 pump2ON <= #23.pump2ON
#27 startDrive <= #23.startDrive
_END_CFC_
(* the same logic as Structured Text *)
(* Блок объединяет в себе RichTwoPumpManager и TwoPumpOneDriveModule. / Дополнительно реализована авария от частотного преобразователя, приходящая / на вход аварии от насоса, контактор которого сейчас включен. / Если при включенном контакторе первого насоса произойдет авария, которая / будет выдана частотным преобразователем, то система отключится и попробует перезапуститься / со вторым насосом и наоборот. / Если после перезапуска снова произойдет авария, при этом авария первого насоса не будет снята, / система остановится. *)
richTwoPumpManager(start := start, setPump1main := setPump1main, setPump2main := setPump2main, setByCounter := setByCounter, setByWorkTime := setByWorkTime, resetPump1counter := resetPump1Counter, resetPump2counter := resetPump2Counter, resetWorkTimePump1 := resetWorkTimePump1, resetWorkTimePump2 := resetWorkTimePump2, startPump1man := startPump1man, startPump2man := startPump2man, stop := stop, resetAlarms := resetAlarms, delayRepeatedStartTime := delayRepeatedStartTime, alarmPump1input := alarmPump1input OR (pump1ON AND driveAlarm), alarmPump2input := (driveAlarm AND pump2ON) OR alarmPump2input);
regimePump1Main := richTwoPumpManager.regimePump1Main;
regimePump2Main := richTwoPumpManager.regimePump2Main;
regimeByCounter := richTwoPumpManager.regimeByCounter;
regimeByWorkTime := richTwoPumpManager.regimeByWorkTime;
counterPump1 := richTwoPumpManager.counterPump1;
counterPump2 := richTwoPumpManager.counterPump2;
daysPump1 := richTwoPumpManager.daysPump1;
hoursPump1 := richTwoPumpManager.hoursPump1;
minutesPump1 := richTwoPumpManager.minutesPump1;
secondsPump1 := richTwoPumpManager.secondsPump1;
daysPump2 := richTwoPumpManager.daysPump2;
hoursPump2 := richTwoPumpManager.hoursPump2;
minutesPump2 := richTwoPumpManager.minutesPump2;
secondsPump2 := richTwoPumpManager.secondsPump2;
nextStartP1timer := richTwoPumpManager.nextStartP1timer;
nextStartP2timer := richTwoPumpManager.nextStartP2timer;
alarmPump1output := richTwoPumpManager.alarmPump1output;
alarmPump2output := richTwoPumpManager.alarmPump2output;
twoPumpOneDriveModule(startPump1 := richTwoPumpManager.pump1starter, startPump2 := richTwoPumpManager.pump2starter);
drivePower := twoPumpOneDriveModule.drivePower;
pump1ON := twoPumpOneDriveModule.pump1ON;
pump2ON := twoPumpOneDriveModule.pump2ON;
startDrive := twoPumpOneDriveModule.startDrive;
END_FUNCTION_BLOCK

(* POU TwoPumpOneDriveModule, CFC *)
FUNCTION_BLOCK TwoPumpOneDriveModule
VAR_INPUT
	startPump1: BOOL;		(*Входящий сигнал на запуск первого насоса.*)
	startPump2: BOOL;		(*Входящий сигнал на запуск второго насоса.*)
END_VAR
VAR_OUTPUT
	drivePower: BOOL;		(*Выход управления контактором питания ЧРП.*)
	pump1ON: BOOL;		(*Выход управления контактором питания насоса 1.*)
	pump2ON: BOOL;		(*Выход управления контактором питания насоса 2.*)
	startDrive: BOOL;		(*Сигнал пуск в ЧРП.*)
END_VAR
VAR
	pump1Off: BOOL;		(*Сигнал на отключение контактора насоса 1.*)
	pump2Off: BOOL;		(*Сигнал на отключение контактора насоса 2.*)
	startP1trig: R_TRIG;		(*Триггер переднего фронта сигнала на запуск насоса 1.*)
	startP2trig: R_TRIG;		(*Триггер переднего фронта сигнала на запуск насоса 2.*)
	ifP1on: IfBOOL;		(*Блок отправляет сигнал на запуск насоса 1 по одной
			из двух веток в зависимости от состояния ключа.*)
	ifP2on: IfBOOL;		(*Блок отправляет сигнал на запуск насоса 2 по одной
			из двух веток в зависимости от состояния ключа.*)
	startDriveDelay: TON;		(*Блок задержки подачи сигнала на включение ЧРП.*)
	stopDriveTrig: F_TRIG;		(*Триггер спада сигнала на включение насоса 1 или 2 для
			снятия сигнала пуск в ЧРП.*)
	p1ONdelay: TON;		(*Задержка на включение контактора насоса 1.*)
	p2ONdelay: TON;		(*Задержка на включение контактора насоса 2.*)
	startDriveTrig: RS;		(*RS триггер сигнала пуск в ЧРП.*)
	p1powerTrig: RS;		(*RS триггер включения контактора насоса 1.*)
	p2powerTrig: RS;		(*RS триггер включения контактора насоса 2.*)
	offP1delayTrig: RS;		(*RS триггер сигнала на отключение контактора насоса 1.*)
	offP2delayTrig: RS;		(*RS триггер сигнала на отключение контактора насоса 2.*)
	offPowerDelay: TOF;		(*Блок управления временем выключения контактора питания ЧРП.*)
	offP2delay: TON;		(*Задержка выключения контактора насоса 1.*)
	offP1delay: TON;		(*Задержка выключения контактора насоса 2.*)
	fastStart: BOOL;		(*Быстрый сигнал на пуск в ЧРП, если не надо переключать
			контакторы.*)
END_VAR
VAR (* helpers for the ST form of the networks *)
	_t160 : BOOL;
END_VAR
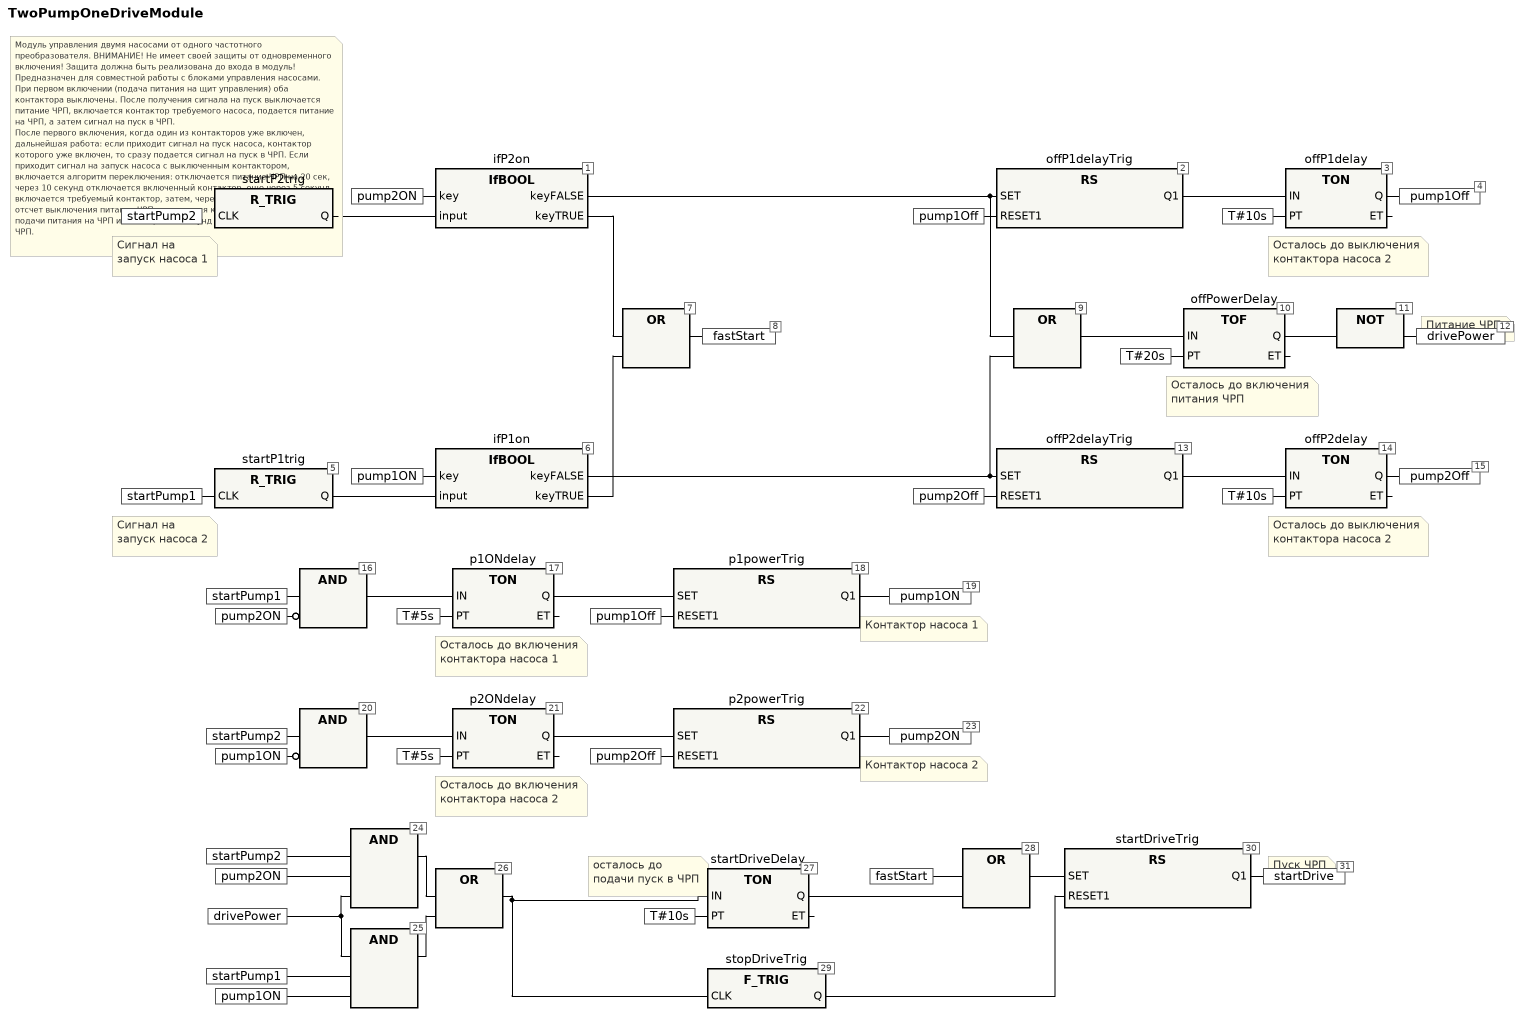
_CFC_ (* Continuous Function Chart, elements in execution order *)
(* Модуль управления двумя насосами от одного частотного преобразователя. ВНИМАНИЕ! Не имеет своей защиты от одновременного включения! Защита должна быть реализована до входа в модуль! Предназначен для совместной работы с блоками управления насосами. / При первом включении (подача питания на щит управления) оба контактора выключены. После получения сигнала на пуск выключается питание ЧРП, включается контактор требуемого насоса, подается питание на ЧРП, а затем сигнал на пуск в ЧРП. / После первого включения, когда один из контакторов уже включен, дальнейшая работа: если приходит сигнал на пуск насоса, контактор которого уже включен, то сразу подается сигнал на пуск в ЧРП. Если приходит сигнал на запуск насоса с выключенным контактором, / включается алгоритм переключения: отключается питание ЧРП на 20 сек, через 10 секунд отключается включенный контактор, еще через 5 секунд включается требуемый контактор, затем, через 5 секунд, заканчивается отсчет выключения питания ЧРП, включается контактор / подачи питания на ЧРП и еще через 10 секунд подается питание на пуск в ЧРП. *)
(* Сигнал на / запуск насоса 2 *)
(* Сигнал на / запуск насоса 1 *)
(* Контактор насоса 1 *)
(* Осталось до включения / контактора насоса 1 *)
(* Контактор насоса 2 *)
(* Осталось до выключения / контактора насоса 2 *)
(* Осталось до включения / питания ЧРП *)
(* Питание ЧРП. *)
(* Осталось до включения / контактора насоса 2 *)
(* Осталось до выключения / контактора насоса 2 *)
(* осталось до / подачи пуск в ЧРП *)
(* Пуск ЧРП *)
#0 startP2trig:R_TRIG(CLK: startPump2)
#1 ifP2on:IfBOOL(key: pump2ON, input: #0.Q)
#2 offP1delayTrig:RS(SET: #1.keyFALSE, RESET1: pump1Off)
#3 offP1delay:TON(IN: #2.Q1, PT: T#10s)
#4 pump1Off <= #3.Q
#5 startP1trig:R_TRIG(CLK: startPump1)
#6 ifP1on:IfBOOL(key: pump1ON, input: #5.Q)
#7 OR(#1.keyTRUE, #6.keyTRUE)
#8 fastStart <= #7
#9 OR(#1.keyFALSE, #6.keyFALSE)
#10 offPowerDelay:TOF(IN: #9, PT: T#20s)
#11 NOT(#10.Q)
#12 drivePower <= #11
#13 offP2delayTrig:RS(SET: #6.keyFALSE, RESET1: pump2Off)
#14 offP2delay:TON(IN: #13.Q1, PT: T#10s)
#15 pump2Off <= #14.Q
#16 AND(startPump1, NOT pump2ON)
#17 p1ONdelay:TON(IN: #16, PT: T#5s)
#18 p1powerTrig:RS(SET: #17.Q, RESET1: pump1Off)
#19 pump1ON <= #18.Q1
#20 AND(startPump2, NOT pump1ON)
#21 p2ONdelay:TON(IN: #20, PT: T#5s)
#22 p2powerTrig:RS(SET: #21.Q, RESET1: pump2Off)
#23 pump2ON <= #22.Q1
#24 AND(startPump2, pump2ON, drivePower)
#25 AND(drivePower, startPump1, pump1ON)
#26 OR(#24, #25)
#27 startDriveDelay:TON(IN: #26, PT: T#10s)
#28 OR(fastStart, #27.Q)
#29 stopDriveTrig:F_TRIG(CLK: #26)
#30 startDriveTrig:RS(SET: #28, RESET1: #29.Q)
#31 startDrive <= #30.Q1
_END_CFC_
(* the same logic as Structured Text *)
(* Модуль управления двумя насосами от одного частотного преобразователя. ВНИМАНИЕ! Не имеет своей защиты от одновременного включения! Защита должна быть реализована до входа в модуль! Предназначен для совместной работы с блоками управления насосами. / При первом включении (подача питания на щит управления) оба контактора выключены. После получения сигнала на пуск выключается питание ЧРП, включается контактор требуемого насоса, подается питание на ЧРП, а затем сигнал на пуск в ЧРП. / После первого включения, когда один из контакторов уже включен, дальнейшая работа: если приходит сигнал на пуск насоса, контактор которого уже включен, то сразу подается сигнал на пуск в ЧРП. Если приходит сигнал на запуск насоса с выключенным контактором, / включается алгоритм переключения: отключается питание ЧРП на 20 сек, через 10 секунд отключается включенный контактор, еще через 5 секунд включается требуемый контактор, затем, через 5 секунд, заканчивается отсчет выключения питания ЧРП, включается контактор / подачи питания на ЧРП и еще через 10 секунд подается питание на пуск в ЧРП. *)
(* Сигнал на / запуск насоса 2 *)
(* Сигнал на / запуск насоса 1 *)
(* Контактор насоса 1 *)
(* Осталось до включения / контактора насоса 1 *)
(* Контактор насоса 2 *)
(* Осталось до выключения / контактора насоса 2 *)
(* Осталось до включения / питания ЧРП *)
(* Питание ЧРП. *)
(* Осталось до включения / контактора насоса 2 *)
(* Осталось до выключения / контактора насоса 2 *)
(* осталось до / подачи пуск в ЧРП *)
(* Пуск ЧРП *)
startP2trig(CLK := startPump2);
ifP2on(key := pump2ON, input := startP2trig.Q);
offP1delayTrig(SET := ifP2on.keyFALSE, RESET1 := pump1Off);
offP1delay(IN := offP1delayTrig.Q1, PT := T#10s);
pump1Off := offP1delay.Q;
startP1trig(CLK := startPump1);
ifP1on(key := pump1ON, input := startP1trig.Q);
fastStart := ifP2on.keyTRUE OR ifP1on.keyTRUE;
offPowerDelay(IN := ifP2on.keyFALSE OR ifP1on.keyFALSE, PT := T#20s);
drivePower := NOT offPowerDelay.Q;
offP2delayTrig(SET := ifP1on.keyFALSE, RESET1 := pump2Off);
offP2delay(IN := offP2delayTrig.Q1, PT := T#10s);
pump2Off := offP2delay.Q;
p1ONdelay(IN := startPump1 AND NOT pump2ON, PT := T#5s);
p1powerTrig(SET := p1ONdelay.Q, RESET1 := pump1Off);
pump1ON := p1powerTrig.Q1;
p2ONdelay(IN := startPump2 AND NOT pump1ON, PT := T#5s);
p2powerTrig(SET := p2ONdelay.Q, RESET1 := pump2Off);
pump2ON := p2powerTrig.Q1;
_t160 := (startPump2 AND pump2ON AND drivePower) OR (drivePower AND startPump1 AND pump1ON);
startDriveDelay(IN := _t160, PT := T#10s);
stopDriveTrig(CLK := _t160);
startDriveTrig(SET := fastStart OR startDriveDelay.Q, RESET1 := stopDriveTrig.Q);
startDrive := startDriveTrig.Q1;
END_FUNCTION_BLOCK
